ABB RAPID module: ReplayTargets_v11.mod

MODULE ReplayTargets_v11
    ! Generated from tests_v11.csv and success_v11.csv.
    ! Target names include testId. B* variants and configuration variables include testId and confId.

    ! Robtargets and jointtargets for replay
    CONST robtarget rA_t1 := [[1867.5,0,1823],[2.18557E-8,0,-1,0],[0,0,0,0],[9E+09,9E+09,9E+09,9E+09,9E+09,9E+09]];
    CONST robtarget rB_t1 := [[1165.98,1084.18,2334.34],[0.470302,-0.608433,0.138324,-0.624093],[0,3,3,0],[9E+09,9E+09,9E+09,9E+09,9E+09,9E+09]];
    CONST robtarget rB_t1_c5 := [[1165.98,1084.18,2334.34],[0.470302,-0.608433,0.138324,-0.624093],[0,0,0,0],[9E+09,9E+09,9E+09,9E+09,9E+09,9E+09]];
    CONST robtarget rB_t1_c6 := [[1165.98,1084.18,2334.34],[0.470302,-0.608433,0.138324,-0.624093],[0,4,0,0],[9E+09,9E+09,9E+09,9E+09,9E+09,9E+09]];
    CONST jointtarget jA_t1 := [[0,-2.3802E-6,7.25062E-7,0,90,0],[9E+09,9E+09,9E+09,9E+09,9E+09,9E+09]];
    CONST jointtarget jB_t1 := [[45.0004,-17.5512,3.9027,270,20.2686,315],[9E+09,9E+09,9E+09,9E+09,9E+09,9E+09]];
    CONST jointtarget jBseed_t1 := [[45.0004,-17.5512,3.9027,270,20.2686,315],[9E+09,9E+09,9E+09,9E+09,9E+09,9E+09]];

    CONST robtarget rA_t4 := [[-1793.05,1763.6,2052.64],[0.337402,0.281183,-0.557431,-0.704533],[1,-3,-1,0],[9E+09,9E+09,9E+09,9E+09,9E+09,9E+09]];
    CONST robtarget rB_t4 := [[-0.00867415,1613.24,1410.95],[0.623931,-0.332722,0.332726,0.623939],[1,-2,-2,0],[9E+09,9E+09,9E+09,9E+09,9E+09,9E+09]];
    CONST robtarget rB_t4_c1 := [[-0.00867415,1613.24,1410.95],[0.623931,-0.332722,0.332726,0.623939],[0,-4,-4,0],[9E+09,9E+09,9E+09,9E+09,9E+09,9E+09]];
    CONST robtarget rB_t4_c4 := [[-0.00867415,1613.24,1410.95],[0.623931,-0.332722,0.332726,0.623939],[0,-4,0,0],[9E+09,9E+09,9E+09,9E+09,9E+09,9E+09]];
    CONST jointtarget jA_t4 := [[134.999,27.2488,-32.8513,-225.001,10.1755,-45.0007],[9E+09,9E+09,9E+09,9E+09,9E+09,9E+09]];
    CONST jointtarget jB_t4 := [[90.0003,-18.1701,41.0059,-180,56.6967,-180],[9E+09,9E+09,9E+09,9E+09,9E+09,9E+09]];
    CONST jointtarget jBseed_t4 := [[90.0003,-18.1701,41.0059,-180,56.6967,-180],[9E+09,9E+09,9E+09,9E+09,9E+09,9E+09]];

    CONST robtarget rA_t7 := [[2738.04,83.3778,1374.99],[0.204279,-0.875639,-0.176726,-0.400366],[0,0,-3,0],[9E+09,9E+09,9E+09,9E+09,9E+09,9E+09]];
    CONST robtarget rB_t7 := [[2056.76,0.0250541,368.189],[0.572435,-0.30037,0.725174,-0.237103],[0,-2,-3,0],[9E+09,9E+09,9E+09,9E+09,9E+09,9E+09]];
    CONST robtarget rB_t7_c1 := [[2056.76,0.0250541,368.189],[0.572435,-0.30037,0.725174,-0.237103],[0,-4,-4,0],[9E+09,9E+09,9E+09,9E+09,9E+09,9E+09]];
    CONST robtarget rB_t7_c2 := [[2056.76,0.0250541,368.189],[0.572435,-0.30037,0.725174,-0.237103],[0,0,-4,0],[9E+09,9E+09,9E+09,9E+09,9E+09,9E+09]];
    CONST jointtarget jA_t7 := [[2.67622E-5,42.2346,-33.9622,45,44.9153,-225],[9E+09,9E+09,9E+09,9E+09,9E+09,9E+09]];
    CONST jointtarget jB_t7 := [[0.000739783,31.9694,26.4257,-179.999,44.9684,-224.999],[9E+09,9E+09,9E+09,9E+09,9E+09,9E+09]];
    CONST jointtarget jBseed_t7 := [[0.000739982,31.9694,26.4257,-179.999,44.9684,-224.999],[9E+09,9E+09,9E+09,9E+09,9E+09,9E+09]];

    CONST robtarget rA_t9 := [[-1368.98,-1368.96,2775.29],[0.617027,1.37404E-6,-0.488433,0.617018],[-2,-3,-4,0],[9E+09,9E+09,9E+09,9E+09,9E+09,9E+09]];
    CONST robtarget rB_t9 := [[-127.824,-1431.05,1500.85],[0.635695,0.309679,-0.685821,0.172164],[-2,-2,2,0],[9E+09,9E+09,9E+09,9E+09,9E+09,9E+09]];
    CONST robtarget rB_t9_c5 := [[-127.824,-1431.05,1500.85],[0.635695,0.309679,-0.685821,0.172164],[0,0,0,0],[9E+09,9E+09,9E+09,9E+09,9E+09,9E+09]];
    CONST jointtarget jA_t9 := [[-135,10.9152,-39.5999,-180,2.84006,-315],[9E+09,9E+09,9E+09,9E+09,9E+09,9E+09]];
    CONST jointtarget jB_t9 := [[-90.0007,-29.3912,41.2717,-90.0007,49.9344,269.999],[9E+09,9E+09,9E+09,9E+09,9E+09,9E+09]];
    CONST jointtarget jBseed_t9 := [[-90.0007,-29.3912,41.2717,-90.0007,49.9344,269.999],[9E+09,9E+09,9E+09,9E+09,9E+09,9E+09]];

    CONST robtarget rA_t12 := [[1027.41,1027.39,1309.98],[0.608549,-0.561103,0.561098,-7.84079E-6],[0,-3,1,0],[9E+09,9E+09,9E+09,9E+09,9E+09,9E+09]];
    CONST robtarget rB_t12 := [[-1587.99,1648.05,1389.04],[0.657658,-0.705427,-0.212225,0.15754],[1,-2,-4,0],[9E+09,9E+09,9E+09,9E+09,9E+09,9E+09]];
    CONST robtarget rB_t12_c4 := [[-1587.99,1648.05,1389.04],[0.657658,-0.705427,-0.212225,0.15754],[0,-4,0,0],[9E+09,9E+09,9E+09,9E+09,9E+09,9E+09]];
    CONST robtarget rB_t12_c5 := [[-1587.99,1648.05,1389.04],[0.657658,-0.705427,-0.212225,0.15754],[0,0,0,0],[9E+09,9E+09,9E+09,9E+09,9E+09,9E+09]];
    CONST jointtarget jA_t12 := [[44.9995,-30.1419,48.0401,-180.001,2.86752,134.999],[9E+09,9E+09,9E+09,9E+09,9E+09,9E+09]];
    CONST jointtarget jB_t12 := [[135,14.8265,5.47776,-135,21.0743,-315],[9E+09,9E+09,9E+09,9E+09,9E+09,9E+09]];
    CONST jointtarget jBseed_t12 := [[135,14.8265,5.47777,-135,21.0743,-315],[9E+09,9E+09,9E+09,9E+09,9E+09,9E+09]];

    CONST robtarget rA_t16 := [[-9.45088,2636.5,793.339],[0.463779,-0.798683,-0.345911,-0.165411],[0,-4,-3,0],[9E+09,9E+09,9E+09,9E+09,9E+09,9E+09]];
    CONST robtarget rB_t16 := [[1243.34,1193.68,2340.57],[0.833225,-0.325403,0.441958,-0.0672477],[0,-2,-3,0],[9E+09,9E+09,9E+09,9E+09,9E+09,9E+09]];
    CONST robtarget rB_t16_c2 := [[1243.34,1193.68,2340.57],[0.833225,-0.325403,0.441958,-0.0672477],[0,0,-4,0],[9E+09,9E+09,9E+09,9E+09,9E+09,9E+09]];
    CONST jointtarget jA_t16 := [[89.9999,41.6852,-10.6259,-270,3.24656,-225],[9E+09,9E+09,9E+09,9E+09,9E+09,9E+09]];
    CONST jointtarget jB_t16 := [[45.0001,-11.4243,-0.148013,-135,17.304,-270],[9E+09,9E+09,9E+09,9E+09,9E+09,9E+09]];
    CONST jointtarget jBseed_t16 := [[45.0001,-11.4243,-0.148018,-135,17.304,-270],[9E+09,9E+09,9E+09,9E+09,9E+09,9E+09]];

    CONST robtarget rA_t19 := [[-102.211,-1856.03,1361.59],[0.589306,0.574164,0.0334011,-0.567397],[-1,2,-2,0],[9E+09,9E+09,9E+09,9E+09,9E+09,9E+09]];
    CONST robtarget rB_t19 := [[1138.52,-1275.9,-60.9308],[0.259666,0.355191,0.770598,-0.461076],[-1,2,-3,0],[9E+09,9E+09,9E+09,9E+09,9E+09,9E+09]];
    CONST robtarget rB_t19_c2 := [[1138.52,-1275.9,-60.9308],[0.259666,0.355191,0.770598,-0.461076],[0,0,-4,0],[9E+09,9E+09,9E+09,9E+09,9E+09,9E+09]];
    CONST jointtarget jA_t19 := [[-89.9992,-3.43333,28.826,225.001,59.9707,-179.999],[9E+09,9E+09,9E+09,9E+09,9E+09,9E+09]];
    CONST jointtarget jB_t19 := [[-45.0008,43.0879,35.2809,224.999,55.327,-225.001],[9E+09,9E+09,9E+09,9E+09,9E+09,9E+09]];
    CONST jointtarget jBseed_t19 := [[-45.0008,43.0879,35.2809,224.999,55.327,-225.001],[9E+09,9E+09,9E+09,9E+09,9E+09,9E+09]];

    CONST robtarget rA_t22 := [[972.378,-908.4,1704.11],[0.389489,-0.323377,0.531814,-0.678896],[-1,1,-3,0],[9E+09,9E+09,9E+09,9E+09,9E+09,9E+09]];
    CONST robtarget rB_t22 := [[958.385,1131.9,1340.89],[0.368991,-0.50086,0.597944,0.505419],[0,0,2,0],[9E+09,9E+09,9E+09,9E+09,9E+09,9E+09]];
    CONST robtarget rB_t22_c5 := [[958.385,1131.9,1340.89],[0.368991,-0.50086,0.597944,0.505419],[0,0,0,0],[9E+09,9E+09,9E+09,9E+09,9E+09,9E+09]];
    CONST jointtarget jA_t22 := [[-45.0004,-38.8031,41.6208,135,22.53,-225],[9E+09,9E+09,9E+09,9E+09,9E+09,9E+09]];
    CONST jointtarget jB_t22 := [[44.9997,-25.3517,43.9894,89.9997,47.2848,270],[9E+09,9E+09,9E+09,9E+09,9E+09,9E+09]];
    CONST jointtarget jBseed_t22 := [[44.9997,-25.3517,43.9894,89.9997,47.2848,270],[9E+09,9E+09,9E+09,9E+09,9E+09,9E+09]];

    CONST robtarget rA_t23 := [[958.385,1131.9,1340.89],[0.368991,-0.50086,0.597944,0.505419],[0,0,2,0],[9E+09,9E+09,9E+09,9E+09,9E+09,9E+09]];
    CONST robtarget rB_t23 := [[-1885.02,1961.47,581.585],[0.429751,-0.871071,0.0769368,0.22501],[1,-2,-4,0],[9E+09,9E+09,9E+09,9E+09,9E+09,9E+09]];
    CONST robtarget rB_t23_c6 := [[-1885.02,1961.47,581.585],[0.429751,-0.871071,0.0769368,0.22501],[0,4,0,0],[9E+09,9E+09,9E+09,9E+09,9E+09,9E+09]];
    CONST jointtarget jA_t23 := [[44.9997,-25.3517,43.9894,89.9997,47.2848,270],[9E+09,9E+09,9E+09,9E+09,9E+09,9E+09]];
    CONST jointtarget jB_t23 := [[134.999,51.3205,-17.3031,-90.0009,18.8714,-315.001],[9E+09,9E+09,9E+09,9E+09,9E+09,9E+09]];
    CONST jointtarget jBseed_t23 := [[134.999,51.3205,-17.3031,-90.0009,18.8714,-315.001],[9E+09,9E+09,9E+09,9E+09,9E+09,9E+09]];

    CONST robtarget rA_t27 := [[-855.452,855.457,3218.91],[0.702987,0.107827,-1.23278E-6,0.702981],[1,1,1,0],[9E+09,9E+09,9E+09,9E+09,9E+09,9E+09]];
    CONST robtarget rB_t27 := [[0.00862806,893.795,2601.28],[0.375694,-0.0727351,-0.175609,-0.907042],[0,1,-1,0],[9E+09,9E+09,9E+09,9E+09,9E+09,9E+09]];
    CONST robtarget rB_t27_c5 := [[0.00862806,893.795,2601.28],[0.375694,-0.0727351,-0.175609,-0.907042],[0,0,0,0],[9E+09,9E+09,9E+09,9E+09,9E+09,9E+09]];
    CONST robtarget rB_t27_c8 := [[0.00862806,893.795,2601.28],[0.375694,-0.0727351,-0.175609,-0.907042],[0,0,4,0],[9E+09,9E+09,9E+09,9E+09,9E+09,9E+09]];
    CONST jointtarget jA_t27 := [[135,0.679351,-47.5347,180,55.5248,135],[9E+09,9E+09,9E+09,9E+09,9E+09,9E+09]];
    CONST jointtarget jB_t27 := [[89.9994,-41.2421,11.8296,179.999,38.673,-45.0006],[9E+09,9E+09,9E+09,9E+09,9E+09,9E+09]];
    CONST jointtarget jBseed_t27 := [[89.9994,-41.2421,11.8296,179.999,38.6731,-45.0006],[9E+09,9E+09,9E+09,9E+09,9E+09,9E+09]];

    CONST robtarget rA_t28 := [[0.00862806,893.795,2601.28],[0.375694,-0.0727351,-0.175609,-0.907042],[0,1,-1,0],[9E+09,9E+09,9E+09,9E+09,9E+09,9E+09]];
    CONST robtarget rB_t28 := [[66.616,1510.09,107.25],[0.0864039,-0.670046,-0.632294,-0.379179],[0,-2,3,0],[9E+09,9E+09,9E+09,9E+09,9E+09,9E+09]];
    CONST robtarget rB_t28_c5 := [[66.616,1510.09,107.25],[0.0864039,-0.670046,-0.632294,-0.379179],[0,0,0,0],[9E+09,9E+09,9E+09,9E+09,9E+09,9E+09]];
    CONST jointtarget jA_t28 := [[89.9994,-41.2421,11.8296,179.999,38.673,-45.0006],[9E+09,9E+09,9E+09,9E+09,9E+09,9E+09]];
    CONST jointtarget jB_t28 := [[89.9998,26.78,48.5241,-135,34.3388,315],[9E+09,9E+09,9E+09,9E+09,9E+09,9E+09]];
    CONST jointtarget jBseed_t28 := [[89.9998,26.78,48.5241,-135,34.3388,315],[9E+09,9E+09,9E+09,9E+09,9E+09,9E+09]];

    CONST robtarget rA_t31 := [[0.0247556,-2099.99,69.6706],[0.317201,0.631961,-0.63197,0.317209],[-1,-2,0,0],[9E+09,9E+09,9E+09,9E+09,9E+09,9E+09]];
    CONST robtarget rB_t31 := [[1527.9,-1527.94,1319.85],[0.854699,0.367072,0.36708,-1.01895E-5],[-1,1,-2,0],[9E+09,9E+09,9E+09,9E+09,9E+09,9E+09]];
    CONST robtarget rB_t31_c1 := [[1527.9,-1527.94,1319.85],[0.854699,0.367072,0.36708,-1.01895E-5],[0,-4,-4,0],[9E+09,9E+09,9E+09,9E+09,9E+09,9E+09]];
    CONST robtarget rB_t31_c4 := [[1527.9,-1527.94,1319.85],[0.854699,0.367072,0.36708,-1.01895E-5],[0,-4,0,0],[9E+09,9E+09,9E+09,9E+09,9E+09,9E+09]];
    CONST jointtarget jA_t31 := [[-89.9993,44.4173,19.4034,-179.999,27.1279,0.000700849],[9E+09,9E+09,9E+09,9E+09,9E+09,9E+09]];
    CONST jointtarget jB_t31 := [[-45.0007,11.4902,15.5232,179.999,54.4664,-135.001],[9E+09,9E+09,9E+09,9E+09,9E+09,9E+09]];
    CONST jointtarget jBseed_t31 := [[-45.0007,11.4902,15.5232,179.999,54.4664,-135.001],[9E+09,9E+09,9E+09,9E+09,9E+09,9E+09]];

    CONST robtarget rA_t37 := [[-1966.29,1997.86,669.131],[0.118201,0.309457,-0.836468,-0.436563],[1,-1,1,0],[9E+09,9E+09,9E+09,9E+09,9E+09,9E+09]];
    CONST robtarget rB_t37 := [[2614.3,138.194,1907.14],[0.237671,0.177553,0.665957,0.684463],[0,1,4,0],[9E+09,9E+09,9E+09,9E+09,9E+09,9E+09]];
    CONST robtarget rB_t37_c5 := [[2614.3,138.194,1907.14],[0.237671,0.177553,0.665957,0.684463],[0,0,0,0],[9E+09,9E+09,9E+09,9E+09,9E+09,9E+09]];
    CONST jointtarget jA_t37 := [[135.001,53.3164,-24.4761,-44.9994,10.9098,135.001],[9E+09,9E+09,9E+09,9E+09,9E+09,9E+09]];
    CONST jointtarget jB_t37 := [[0.000991918,37.2063,-42.3057,90.001,55.8159,360.001],[9E+09,9E+09,9E+09,9E+09,9E+09,9E+09]];
    CONST jointtarget jBseed_t37 := [[0.000991821,37.2063,-42.3057,90.001,55.8159,360.001],[9E+09,9E+09,9E+09,9E+09,9E+09,9E+09]];

    CONST robtarget rA_t40 := [[2042.82,2042.82,1269.08],[2.13329E-8,0.491803,0.491803,0.718512],[0,2,3,0],[9E+09,9E+09,9E+09,9E+09,9E+09,9E+09]];
    CONST robtarget rB_t40 := [[2226.68,51.0258,2546.48],[0.890874,-0.128724,0.42641,0.0891495],[0,-3,-2,0],[9E+09,9E+09,9E+09,9E+09,9E+09,9E+09]];
    CONST robtarget rB_t40_c8 := [[2226.68,51.0258,2546.48],[0.890874,-0.128724,0.42641,0.0891495],[0,0,4,0],[9E+09,9E+09,9E+09,9E+09,9E+09,9E+09]];
    CONST jointtarget jA_t40 := [[45,49.2001,-36.7553,180,14.3083,315],[9E+09,9E+09,9E+09,9E+09,9E+09,9E+09]];
    CONST jointtarget jB_t40 := [[0.000737447,21.2244,-41.8256,-224.999,25.5861,-134.999],[9E+09,9E+09,9E+09,9E+09,9E+09,9E+09]];
    CONST jointtarget jBseed_t40 := [[0.00073748,21.2244,-41.8256,-224.999,25.5861,-134.999],[9E+09,9E+09,9E+09,9E+09,9E+09,9E+09]];

    CONST robtarget rA_t46 := [[315.105,315.107,2762.98],[0.664534,5.18351E-7,0.341732,0.66454],[0,-2,-2,0],[9E+09,9E+09,9E+09,9E+09,9E+09,9E+09]];
    CONST robtarget rB_t46 := [[1363.27,1399.66,1627.46],[0.295621,-0.697087,-0.341342,-0.556923],[0,-3,-3,0],[9E+09,9E+09,9E+09,9E+09,9E+09,9E+09]];
    CONST robtarget rB_t46_c1 := [[1363.27,1399.66,1627.46],[0.295621,-0.697087,-0.341342,-0.556923],[0,-4,-4,0],[9E+09,9E+09,9E+09,9E+09,9E+09,9E+09]];
    CONST robtarget rB_t46_c2 := [[1363.27,1399.66,1627.46],[0.295621,-0.697087,-0.341342,-0.556923],[0,0,-4,0],[9E+09,9E+09,9E+09,9E+09,9E+09,9E+09]];
    CONST jointtarget jA_t46 := [[45.0002,-51.9395,4.53749,-180,2.63314,-135],[9E+09,9E+09,9E+09,9E+09,9E+09,9E+09]];
    CONST jointtarget jB_t46 := [[45.0007,-4.25367,16.2215,-269.999,8.85525,-269.999],[9E+09,9E+09,9E+09,9E+09,9E+09,9E+09]];
    CONST jointtarget jBseed_t46 := [[45.0007,-4.25367,16.2215,-269.999,8.85525,-269.999],[9E+09,9E+09,9E+09,9E+09,9E+09,9E+09]];

    CONST robtarget rA_t50 := [[-1650.69,1788.89,2235.47],[0.742108,-0.354072,-0.189288,-0.53673],[1,-2,3,0],[9E+09,9E+09,9E+09,9E+09,9E+09,9E+09]];
    CONST robtarget rB_t50 := [[44.2638,306.55,3391.36],[0.355804,-0.140867,0.00668765,-0.923859],[0,2,-2,0],[9E+09,9E+09,9E+09,9E+09,9E+09,9E+09]];
    CONST robtarget rB_t50_c7 := [[44.2638,306.55,3391.36],[0.355804,-0.140867,0.00668765,-0.923859],[0,-4,4,0],[9E+09,9E+09,9E+09,9E+09,9E+09,9E+09]];
    CONST jointtarget jA_t50 := [[135.001,29.556,-40.0324,-134.999,55.8782,315.001],[9E+09,9E+09,9E+09,9E+09,9E+09,9E+09]];
    CONST jointtarget jB_t50 := [[89.9996,-20.9717,-47.8442,225,22.0136,-90.0004],[9E+09,9E+09,9E+09,9E+09,9E+09,9E+09]];
    CONST jointtarget jBseed_t50 := [[89.9996,-20.9717,-47.8442,225,22.0136,-90.0004],[9E+09,9E+09,9E+09,9E+09,9E+09,9E+09]];

    CONST robtarget rA_t51 := [[44.2638,306.55,3391.36],[0.355804,-0.140867,0.00668765,-0.923859],[0,2,-2,0],[9E+09,9E+09,9E+09,9E+09,9E+09,9E+09]];
    CONST robtarget rB_t51 := [[2033.92,45.4637,1419.42],[0.577235,0.205402,0.70222,0.362625],[0,1,-1,0],[9E+09,9E+09,9E+09,9E+09,9E+09,9E+09]];
    CONST robtarget rB_t51_c5 := [[2033.92,45.4637,1419.42],[0.577235,0.205402,0.70222,0.362625],[0,0,0,0],[9E+09,9E+09,9E+09,9E+09,9E+09,9E+09]];
    CONST robtarget rB_t51_c8 := [[2033.92,45.4637,1419.42],[0.577235,0.205402,0.70222,0.362625],[0,0,4,0],[9E+09,9E+09,9E+09,9E+09,9E+09,9E+09]];
    CONST jointtarget jA_t51 := [[89.9996,-20.9717,-47.8442,225,22.0136,-90.0004],[9E+09,9E+09,9E+09,9E+09,9E+09,9E+09]];
    CONST jointtarget jB_t51 := [[0.000420681,1.789,18.8479,135,22.6362,-89.9996],[9E+09,9E+09,9E+09,9E+09,9E+09,9E+09]];
    CONST jointtarget jBseed_t51 := [[0.000420515,1.789,18.8479,135,22.6362,-89.9996],[9E+09,9E+09,9E+09,9E+09,9E+09,9E+09]];

    CONST robtarget rA_t53 := [[39.7549,2396.44,2309.29],[0.688612,-0.598908,0.352715,0.206675],[1,-1,-4,0],[9E+09,9E+09,9E+09,9E+09,9E+09,9E+09]];
    CONST robtarget rB_t53 := [[1503.67,-0.0118296,1707.84],[0.639783,0.276074,0.666511,0.264998],[-1,1,-2,0],[9E+09,9E+09,9E+09,9E+09,9E+09,9E+09]];
    CONST robtarget rB_t53_c1 := [[1503.67,-0.0118296,1707.84],[0.639783,0.276074,0.666511,0.264998],[0,-4,-4,0],[9E+09,9E+09,9E+09,9E+09,9E+09,9E+09]];
    CONST jointtarget jA_t53 := [[90.0007,25.6044,-41.7978,-44.9993,19.6881,-359.999],[9E+09,9E+09,9E+09,9E+09,9E+09,9E+09]];
    CONST jointtarget jB_t53 := [[-0.000453216,-28.9554,33.9439,180,2.64412,-135],[9E+09,9E+09,9E+09,9E+09,9E+09,9E+09]];
    CONST jointtarget jBseed_t53 := [[-0.000453108,-28.9554,33.9439,180,2.64412,-135],[9E+09,9E+09,9E+09,9E+09,9E+09,9E+09]];

    CONST robtarget rA_t56 := [[-781.455,-757.26,2911.76],[0.356269,-0.225306,-0.422891,0.802167],[-2,-1,-1,0],[9E+09,9E+09,9E+09,9E+09,9E+09,9E+09]];
    CONST robtarget rB_t56 := [[-1461,-1377.29,2942.46],[0.626638,0.215306,-0.16846,-0.729787],[-2,2,2,0],[9E+09,9E+09,9E+09,9E+09,9E+09,9E+09]];
    CONST robtarget rB_t56_c2 := [[-1461,-1377.29,2942.46],[0.626638,0.215306,-0.16846,-0.729787],[0,0,-4,0],[9E+09,9E+09,9E+09,9E+09,9E+09,9E+09]];
    CONST robtarget rB_t56_c5 := [[-1461,-1377.29,2942.46],[0.626638,0.215306,-0.16846,-0.729787],[0,0,0,0],[9E+09,9E+09,9E+09,9E+09,9E+09,9E+09]];
    CONST jointtarget jA_t56 := [[-135,-23.7587,-15.0853,-45.0001,8.32972,-45.0001],[9E+09,9E+09,9E+09,9E+09,9E+09,9E+09]];
    CONST jointtarget jB_t56 := [[-134.999,34.2473,-77.4173,225.001,30.0943,180.001],[9E+09,9E+09,9E+09,9E+09,9E+09,9E+09]];
    CONST jointtarget jBseed_t56 := [[-134.999,34.2473,-77.4172,225.001,30.0943,180.001],[9E+09,9E+09,9E+09,9E+09,9E+09,9E+09]];

    CONST robtarget rA_t58 := [[-516.819,-387.904,3130.9],[0.270635,0.128291,-0.254314,-0.919578],[-2,2,1,0],[9E+09,9E+09,9E+09,9E+09,9E+09,9E+09]];
    CONST robtarget rB_t58 := [[18.5522,-2972.36,1606.68],[0.550399,0.443924,0.502249,-0.497733],[-1,1,-1,0],[9E+09,9E+09,9E+09,9E+09,9E+09,9E+09]];
    CONST robtarget rB_t58_c8 := [[18.5522,-2972.36,1606.68],[0.550399,0.443924,0.502249,-0.497733],[0,0,4,0],[9E+09,9E+09,9E+09,9E+09,9E+09,9E+09]];
    CONST jointtarget jA_t58 := [[-135.001,-26.8752,-23.6708,224.999,50.524,134.999],[9E+09,9E+09,9E+09,9E+09,9E+09,9E+09]];
    CONST jointtarget jB_t58 := [[-89.9996,59.8242,-65.6776,90.0005,6.37043,-89.9997],[9E+09,9E+09,9E+09,9E+09,9E+09,9E+09]];
    CONST jointtarget jBseed_t58 := [[-89.9996,59.8242,-65.6777,90.0004,6.37043,-89.9996],[9E+09,9E+09,9E+09,9E+09,9E+09,9E+09]];

    CONST robtarget rA_t64 := [[-1515.54,1515.56,1455.6],[0.333635,0.187434,-0.452494,-0.805485],[1,-3,-2,0],[9E+09,9E+09,9E+09,9E+09,9E+09,9E+09]];
    CONST robtarget rB_t64 := [[2573.98,0.0267315,1917.9],[1.18647E-5,-0.542748,4.45635E-6,-0.839896],[0,-2,4,0],[9E+09,9E+09,9E+09,9E+09,9E+09,9E+09]];
    CONST robtarget rB_t64_c4 := [[2573.98,0.0267315,1917.9],[1.18647E-5,-0.542748,4.45635E-6,-0.839896],[0,-4,0,0],[9E+09,9E+09,9E+09,9E+09,9E+09,9E+09]];
    CONST jointtarget jA_t64 := [[135,8.96329,13.5435,-180,53.8548,-90.0005],[9E+09,9E+09,9E+09,9E+09,9E+09,9E+09]];
    CONST jointtarget jB_t64 := [[0.000611133,29.7098,-29.9512,-179.999,24.0168,360.001],[9E+09,9E+09,9E+09,9E+09,9E+09,9E+09]];
    CONST jointtarget jBseed_t64 := [[0.000611133,29.7098,-29.9512,-179.999,24.0168,360.001],[9E+09,9E+09,9E+09,9E+09,9E+09,9E+09]];

    CONST robtarget rA_t66 := [[2907.11,71.3398,1111.81],[0.299575,0.451234,0.640506,0.544421],[0,-3,4,0],[9E+09,9E+09,9E+09,9E+09,9E+09,9E+09]];
    CONST robtarget rB_t66 := [[1282.21,1138.81,-182.246],[0.536967,0.025283,0.842048,0.0445313],[0,-2,-3,0],[9E+09,9E+09,9E+09,9E+09,9E+09,9E+09]];
    CONST robtarget rB_t66_c4 := [[1282.21,1138.81,-182.246],[0.536967,0.025283,0.842048,0.0445313],[0,-4,0,0],[9E+09,9E+09,9E+09,9E+09,9E+09,9E+09]];
    CONST jointtarget jA_t66 := [[0.000451427,52.8733,-38.2867,-270,25.2803,360],[9E+09,9E+09,9E+09,9E+09,9E+09,9E+09]];
    CONST jointtarget jB_t66 := [[45,49.9838,31.7103,-135,59.1723,-180],[9E+09,9E+09,9E+09,9E+09,9E+09,9E+09]];
    CONST jointtarget jBseed_t66 := [[45,49.9838,31.7103,-135,59.1723,-180],[9E+09,9E+09,9E+09,9E+09,9E+09,9E+09]];

    CONST robtarget rA_t67 := [[1282.21,1138.81,-182.246],[0.536967,0.025283,0.842048,0.0445313],[0,-2,-3,0],[9E+09,9E+09,9E+09,9E+09,9E+09,9E+09]];
    CONST robtarget rB_t67 := [[33.2258,843.078,3012.65],[0.865057,-0.313323,0.22989,0.317263],[0,-2,-4,0],[9E+09,9E+09,9E+09,9E+09,9E+09,9E+09]];
    CONST robtarget rB_t67_c2 := [[33.2258,843.078,3012.65],[0.865057,-0.313323,0.22989,0.317263],[0,0,-4,0],[9E+09,9E+09,9E+09,9E+09,9E+09,9E+09]];
    CONST robtarget rB_t67_c3 := [[33.2258,843.078,3012.65],[0.865057,-0.313323,0.22989,0.317263],[0,4,-4,0],[9E+09,9E+09,9E+09,9E+09,9E+09,9E+09]];
    CONST jointtarget jA_t67 := [[45,49.9838,31.7103,-135,59.1723,-180],[9E+09,9E+09,9E+09,9E+09,9E+09,9E+09]];
    CONST jointtarget jB_t67 := [[89.9996,-28.5745,-16.8389,-90.0004,11.4737,-315],[9E+09,9E+09,9E+09,9E+09,9E+09,9E+09]];
    CONST jointtarget jBseed_t67 := [[89.9996,-28.5745,-16.8389,-90.0004,11.4737,-315],[9E+09,9E+09,9E+09,9E+09,9E+09,9E+09]];

    CONST robtarget rA_t68 := [[33.2258,843.078,3012.65],[0.865057,-0.313323,0.22989,0.317263],[0,-2,-4,0],[9E+09,9E+09,9E+09,9E+09,9E+09,9E+09]];
    CONST robtarget rB_t68 := [[1863.94,-1731.5,1359.6],[0.365907,0.552226,0.180387,0.727062],[-1,-3,-1,0],[9E+09,9E+09,9E+09,9E+09,9E+09,9E+09]];
    CONST robtarget rB_t68_c4 := [[1863.94,-1731.5,1359.6],[0.365907,0.552226,0.180387,0.727062],[0,-4,0,0],[9E+09,9E+09,9E+09,9E+09,9E+09,9E+09]];
    CONST jointtarget jA_t68 := [[89.9996,-28.5745,-16.8389,-90.0004,11.4737,-315],[9E+09,9E+09,9E+09,9E+09,9E+09,9E+09]];
    CONST jointtarget jB_t68 := [[-45.0004,30.585,-11.0544,-225,52.4851,-0.000424009],[9E+09,9E+09,9E+09,9E+09,9E+09,9E+09]];
    CONST jointtarget jBseed_t68 := [[-45.0004,30.585,-11.0544,-225,52.4851,-0.00042436],[9E+09,9E+09,9E+09,9E+09,9E+09,9E+09]];

    CONST robtarget rA_t69 := [[1863.94,-1731.5,1359.6],[0.365907,0.552226,0.180387,0.727062],[-1,-3,-1,0],[9E+09,9E+09,9E+09,9E+09,9E+09,9E+09]];
    CONST robtarget rB_t69 := [[90.2483,-604.038,3447.57],[0.635996,0.309007,0.0836555,0.702158],[-1,1,-3,0],[9E+09,9E+09,9E+09,9E+09,9E+09,9E+09]];
    CONST robtarget rB_t69_c4 := [[90.2483,-604.038,3447.57],[0.635996,0.309007,0.0836555,0.702158],[0,-4,0,0],[9E+09,9E+09,9E+09,9E+09,9E+09,9E+09]];
    CONST jointtarget jA_t69 := [[-45.0004,30.585,-11.0544,-225,52.4851,-0.000424009],[9E+09,9E+09,9E+09,9E+09,9E+09,9E+09]];
    CONST jointtarget jB_t69 := [[-89.999,-4.08885,-66.7925,90.001,32.7073,-269.999],[9E+09,9E+09,9E+09,9E+09,9E+09,9E+09]];
    CONST jointtarget jBseed_t69 := [[-89.999,-4.08887,-66.7925,90.001,32.7073,-269.999],[9E+09,9E+09,9E+09,9E+09,9E+09,9E+09]];

    CONST robtarget rA_t72 := [[72.5438,-307.938,3482.9],[0.882145,-0.0280946,0.25871,0.392555],[-1,-3,4,0],[9E+09,9E+09,9E+09,9E+09,9E+09,9E+09]];
    CONST robtarget rB_t72 := [[-1617.38,-1478.51,2678.01],[0.645209,0.274316,-0.69781,-0.14669],[-2,-1,2,0],[9E+09,9E+09,9E+09,9E+09,9E+09,9E+09]];
    CONST robtarget rB_t72_c5 := [[-1617.38,-1478.51,2678.01],[0.645209,0.274316,-0.69781,-0.14669],[0,0,0,0],[9E+09,9E+09,9E+09,9E+09,9E+09,9E+09]];
    CONST jointtarget jA_t72 := [[-89.9997,-5.67095,-71.7875,-225,37.9022,360],[9E+09,9E+09,9E+09,9E+09,9E+09,9E+09]];
    CONST jointtarget jB_t72 := [[-135,34.5695,-72.3707,-44.9996,56.2737,180],[9E+09,9E+09,9E+09,9E+09,9E+09,9E+09]];
    CONST jointtarget jBseed_t72 := [[-135,34.5695,-72.3707,-44.9996,56.2737,180],[9E+09,9E+09,9E+09,9E+09,9E+09,9E+09]];

    CONST robtarget rA_t73 := [[-1617.38,-1478.51,2678.01],[0.645209,0.274316,-0.69781,-0.14669],[-2,-1,2,0],[9E+09,9E+09,9E+09,9E+09,9E+09,9E+09]];
    CONST robtarget rB_t73 := [[1512.76,1682.59,2148.43],[0.670669,-0.609575,-0.292732,-0.304844],[0,0,-3,0],[9E+09,9E+09,9E+09,9E+09,9E+09,9E+09]];
    CONST robtarget rB_t73_c4 := [[1512.76,1682.59,2148.43],[0.670669,-0.609575,-0.292732,-0.304844],[0,-4,0,0],[9E+09,9E+09,9E+09,9E+09,9E+09,9E+09]];
    CONST jointtarget jA_t73 := [[-135,34.5695,-72.3707,-44.9996,56.2737,180],[9E+09,9E+09,9E+09,9E+09,9E+09,9E+09]];
    CONST jointtarget jB_t73 := [[44.9995,16.2365,-23.3018,89.9995,45.9902,-225.001],[9E+09,9E+09,9E+09,9E+09,9E+09,9E+09]];
    CONST jointtarget jBseed_t73 := [[44.9995,16.2365,-23.3018,89.9995,45.9902,-225.001],[9E+09,9E+09,9E+09,9E+09,9E+09,9E+09]];

    CONST robtarget rA_t74 := [[1512.76,1682.59,2148.43],[0.670669,-0.609575,-0.292732,-0.304844],[0,0,-3,0],[9E+09,9E+09,9E+09,9E+09,9E+09,9E+09]];
    CONST robtarget rB_t74 := [[1174.89,-1292.72,-255.154],[0.430425,0.901012,-0.0205942,0.0498761],[-1,-2,-2,0],[9E+09,9E+09,9E+09,9E+09,9E+09,9E+09]];
    CONST robtarget rB_t74_c4 := [[1174.89,-1292.72,-255.154],[0.430425,0.901012,-0.0205942,0.0498761],[0,-4,0,0],[9E+09,9E+09,9E+09,9E+09,9E+09,9E+09]];
    CONST jointtarget jA_t74 := [[44.9995,16.2365,-23.3018,89.9995,45.9902,-225.001],[9E+09,9E+09,9E+09,9E+09,9E+09,9E+09]];
    CONST jointtarget jB_t74 := [[-45.0001,52.7342,28.5125,-135,44.8732,-90.0001],[9E+09,9E+09,9E+09,9E+09,9E+09,9E+09]];
    CONST jointtarget jBseed_t74 := [[-45.0001,52.7342,28.5125,-135,44.8732,-90.0001],[9E+09,9E+09,9E+09,9E+09,9E+09,9E+09]];

    CONST robtarget rA_t79 := [[-816.378,919.561,-368.344],[0.272348,-0.894319,0.350624,0.0555271],[1,-2,-3,0],[9E+09,9E+09,9E+09,9E+09,9E+09,9E+09]];
    CONST robtarget rB_t79 := [[-881.287,1006.84,2597.32],[0.918162,-0.360497,-0.0185053,-0.163334],[1,-2,-5,0],[9E+09,9E+09,9E+09,9E+09,9E+09,9E+09]];
    CONST robtarget rB_t79_c1 := [[-881.287,1006.84,2597.32],[0.918162,-0.360497,-0.0185053,-0.163334],[0,-4,-4,0],[9E+09,9E+09,9E+09,9E+09,9E+09,9E+09]];
    CONST robtarget rB_t79_c4 := [[-881.287,1006.84,2597.32],[0.918162,-0.360497,-0.0185053,-0.163334],[0,-4,0,0],[9E+09,9E+09,9E+09,9E+09,9E+09,9E+09]];
    CONST jointtarget jA_t79 := [[134.999,53.7339,45.3502,-135.001,38.1512,-225.001],[9E+09,9E+09,9E+09,9E+09,9E+09,9E+09]];
    CONST jointtarget jB_t79 := [[135,-21.7334,-0.195621,-135,48.7478,-360],[9E+09,9E+09,9E+09,9E+09,9E+09,9E+09]];
    CONST jointtarget jBseed_t79 := [[135,-21.7334,-0.195625,-135,48.7478,-360],[9E+09,9E+09,9E+09,9E+09,9E+09,9E+09]];

    CONST robtarget rA_t82 := [[-206.925,281.712,3308.39],[0.337776,-0.0648298,-0.253186,-0.904213],[1,3,2,0],[9E+09,9E+09,9E+09,9E+09,9E+09,9E+09]];
    CONST robtarget rB_t82 := [[-869.622,1036.66,1582.29],[0.613039,-0.668325,-0.309037,-0.286392],[1,-1,-1,0],[9E+09,9E+09,9E+09,9E+09,9E+09,9E+09]];
    CONST robtarget rB_t82_c8 := [[-869.622,1036.66,1582.29],[0.613039,-0.668325,-0.309037,-0.286392],[0,0,4,0],[9E+09,9E+09,9E+09,9E+09,9E+09,9E+09]];
    CONST robtarget rB_t82_c9 := [[-869.622,1036.66,1582.29],[0.613039,-0.668325,-0.309037,-0.286392],[0,4,4,0],[9E+09,9E+09,9E+09,9E+09,9E+09,9E+09]];
    CONST jointtarget jA_t82 := [[135.001,-26.4467,-39.0921,270.001,18.4631,180.001],[9E+09,9E+09,9E+09,9E+09,9E+09,9E+09]];
    CONST jointtarget jB_t82 := [[135.001,-35.4485,42.2993,-89.9994,45.0197,-44.9994],[9E+09,9E+09,9E+09,9E+09,9E+09,9E+09]];
    CONST jointtarget jBseed_t82 := [[135.001,-35.4485,42.2993,-89.9994,45.0197,-44.9994],[9E+09,9E+09,9E+09,9E+09,9E+09,9E+09]];

    CONST robtarget rA_t83 := [[-869.622,1036.66,1582.29],[0.613039,-0.668325,-0.309037,-0.286392],[1,-1,-1,0],[9E+09,9E+09,9E+09,9E+09,9E+09,9E+09]];
    CONST robtarget rB_t83 := [[-1630.62,1808.91,1755.18],[0.218749,-0.280556,-0.670403,-0.651151],[1,-1,-2,0],[9E+09,9E+09,9E+09,9E+09,9E+09,9E+09]];
    CONST robtarget rB_t83_c5 := [[-1630.62,1808.91,1755.18],[0.218749,-0.280556,-0.670403,-0.651151],[0,0,0,0],[9E+09,9E+09,9E+09,9E+09,9E+09,9E+09]];
    CONST robtarget rB_t83_c8 := [[-1630.62,1808.91,1755.18],[0.218749,-0.280556,-0.670403,-0.651151],[0,0,4,0],[9E+09,9E+09,9E+09,9E+09,9E+09,9E+09]];
    CONST jointtarget jA_t83 := [[135.001,-35.4485,42.2993,-89.9994,45.0197,-44.9994],[9E+09,9E+09,9E+09,9E+09,9E+09,9E+09]];
    CONST jointtarget jB_t83 := [[135.001,23.3595,-18.4338,-89.9991,49.0353,-134.999],[9E+09,9E+09,9E+09,9E+09,9E+09,9E+09]];
    CONST jointtarget jBseed_t83 := [[135.001,23.3595,-18.4338,-89.9991,49.0353,-134.999],[9E+09,9E+09,9E+09,9E+09,9E+09,9E+09]];

    CONST robtarget rA_t85 := [[1930.15,55.1772,809.731],[0.437101,-0.407513,0.801635,-0.0160386],[-1,-4,2,0],[9E+09,9E+09,9E+09,9E+09,9E+09,9E+09]];
    CONST robtarget rB_t85 := [[1483.71,-1619.15,2708.51],[0.145458,0.140219,-0.512339,0.834679],[-1,-1,3,0],[9E+09,9E+09,9E+09,9E+09,9E+09,9E+09]];
    CONST robtarget rB_t85_c8 := [[1483.71,-1619.15,2708.51],[0.145458,0.140219,-0.512339,0.834679],[0,0,4,0],[9E+09,9E+09,9E+09,9E+09,9E+09,9E+09]];
    CONST jointtarget jA_t85 := [[-0.000696811,9.747,31.1072,-270.001,19.3017,224.999],[9E+09,9E+09,9E+09,9E+09,9E+09,9E+09]];
    CONST jointtarget jB_t85 := [[-44.9998,29.6512,-61.7817,-89.9998,34.9944,315],[9E+09,9E+09,9E+09,9E+09,9E+09,9E+09]];
    CONST jointtarget jBseed_t85 := [[-44.9998,29.6512,-61.7817,-89.9998,34.9944,315],[9E+09,9E+09,9E+09,9E+09,9E+09,9E+09]];

    CONST robtarget rA_t88 := [[1883.97,-1693.67,1011.01],[0.601852,-0.23589,0.760816,-0.0573519],[-1,-4,2,0],[9E+09,9E+09,9E+09,9E+09,9E+09,9E+09]];
    CONST robtarget rB_t88 := [[2631.34,-134.594,1793.98],[0.673616,0.670251,0.215022,0.225323],[0,3,-2,0],[9E+09,9E+09,9E+09,9E+09,9E+09,9E+09]];
    CONST robtarget rB_t88_c5 := [[2631.34,-134.594,1793.98],[0.673616,0.670251,0.215022,0.225323],[0,0,0,0],[9E+09,9E+09,9E+09,9E+09,9E+09,9E+09]];
    CONST jointtarget jA_t88 := [[-45,35.6096,-8.59859,-270,53.6845,225],[9E+09,9E+09,9E+09,9E+09,9E+09,9E+09]];
    CONST jointtarget jB_t88 := [[0.000497925,36.6314,-37.5091,270,53.7156,-179.999],[9E+09,9E+09,9E+09,9E+09,9E+09,9E+09]];
    CONST jointtarget jBseed_t88 := [[0.000497909,36.6314,-37.5091,270,53.7156,-179.999],[9E+09,9E+09,9E+09,9E+09,9E+09,9E+09]];

    CONST robtarget rA_t89 := [[2631.34,-134.594,1793.98],[0.673616,0.670251,0.215022,0.225323],[0,3,-2,0],[9E+09,9E+09,9E+09,9E+09,9E+09,9E+09]];
    CONST robtarget rB_t89 := [[-0.0100308,-1992.85,2351.79],[0.79034,0.612668,1.64E-6,-5.9405E-6],[-2,-3,-2,0],[9E+09,9E+09,9E+09,9E+09,9E+09,9E+09]];
    CONST robtarget rB_t89_c5 := [[-0.0100308,-1992.85,2351.79],[0.79034,0.612668,1.64E-6,-5.9405E-6],[0,0,0,0],[9E+09,9E+09,9E+09,9E+09,9E+09,9E+09]];
    CONST jointtarget jA_t89 := [[0.000497925,36.6314,-37.5091,270,53.7156,-179.999],[9E+09,9E+09,9E+09,9E+09,9E+09,9E+09]];
    CONST jointtarget jB_t89 := [[-90.0003,2.06001,-14.1966,-180,2.29804,-90.0003],[9E+09,9E+09,9E+09,9E+09,9E+09,9E+09]];
    CONST jointtarget jBseed_t89 := [[-90.0003,2.06,-14.1966,-180,2.29804,-90.0003],[9E+09,9E+09,9E+09,9E+09,9E+09,9E+09]];

    CONST robtarget rA_t90 := [[-0.0100308,-1992.85,2351.79],[0.79034,0.612668,1.64E-6,-5.9405E-6],[-2,-3,-2,0],[9E+09,9E+09,9E+09,9E+09,9E+09,9E+09]];
    CONST robtarget rB_t90 := [[1939.65,1939.58,1900.24],[0.407797,-0.829006,0.343384,-0.168931],[0,-1,2,0],[9E+09,9E+09,9E+09,9E+09,9E+09,9E+09]];
    CONST robtarget rB_t90_c5 := [[1939.65,1939.58,1900.24],[0.407797,-0.829006,0.343384,-0.168931],[0,0,0,0],[9E+09,9E+09,9E+09,9E+09,9E+09,9E+09]];
    CONST jointtarget jA_t90 := [[-90.0003,2.06001,-14.1966,-180,2.29804,-90.0003],[9E+09,9E+09,9E+09,9E+09,9E+09,9E+09]];
    CONST jointtarget jB_t90 := [[44.9991,49.6066,-65.1103,-0.000908008,53.1168,269.999],[9E+09,9E+09,9E+09,9E+09,9E+09,9E+09]];
    CONST jointtarget jBseed_t90 := [[44.9991,49.6066,-65.1103,-0.000909421,53.1169,269.999],[9E+09,9E+09,9E+09,9E+09,9E+09,9E+09]];

    CONST robtarget rA_t102 := [[-1948.31,-1917.18,1251.26],[0.646342,0.509608,-0.56543,-0.053206],[-2,2,-1,0],[9E+09,9E+09,9E+09,9E+09,9E+09,9E+09]];
    CONST robtarget rB_t102 := [[-8.1709,-1803.03,1617.76],[0.576867,0.721357,0.282027,-0.259478],[-1,-1,1,0],[9E+09,9E+09,9E+09,9E+09,9E+09,9E+09]];
    CONST robtarget rB_t102_c3 := [[-8.1709,-1803.03,1617.76],[0.576867,0.721357,0.282027,-0.259478],[0,4,-4,0],[9E+09,9E+09,9E+09,9E+09,9E+09,9E+09]];
    CONST jointtarget jA_t102 := [[-135,39.4037,-22.5361,225,10.7523,-89.9997],[9E+09,9E+09,9E+09,9E+09,9E+09,9E+09]];
    CONST jointtarget jB_t102 := [[-89.9998,-12.197,23.7358,-89.9998,2.80709,135],[9E+09,9E+09,9E+09,9E+09,9E+09,9E+09]];
    CONST jointtarget jBseed_t102 := [[-89.9998,-12.197,23.7358,-89.9998,2.80709,135],[9E+09,9E+09,9E+09,9E+09,9E+09,9E+09]];

    CONST robtarget rA_t103 := [[-8.1709,-1803.03,1617.76],[0.576867,0.721357,0.282027,-0.259478],[-1,-1,1,0],[9E+09,9E+09,9E+09,9E+09,9E+09,9E+09]];
    CONST robtarget rB_t103 := [[2153.31,0.0367459,1279.08],[0.0943866,0.700781,0.700775,0.0943998],[0,0,-3,0],[9E+09,9E+09,9E+09,9E+09,9E+09,9E+09]];
    CONST robtarget rB_t103_c5 := [[2153.31,0.0367459,1279.08],[0.0943866,0.700781,0.700775,0.0943998],[0,0,0,0],[9E+09,9E+09,9E+09,9E+09,9E+09,9E+09]];
    CONST jointtarget jA_t103 := [[-89.9998,-12.197,23.7358,-89.9998,2.80709,135],[9E+09,9E+09,9E+09,9E+09,9E+09,9E+09]];
    CONST jointtarget jB_t103 := [[0.00091901,13.5118,5.64439,0.000918909,55.501,-269.999],[9E+09,9E+09,9E+09,9E+09,9E+09,9E+09]];
    CONST jointtarget jBseed_t103 := [[0.000919004,13.5118,5.64439,0.000919004,55.501,-269.999],[9E+09,9E+09,9E+09,9E+09,9E+09,9E+09]];

    CONST robtarget rA_t104 := [[2153.31,0.0367459,1279.08],[0.0943866,0.700781,0.700775,0.0943998],[0,0,-3,0],[9E+09,9E+09,9E+09,9E+09,9E+09,9E+09]];
    CONST robtarget rB_t104 := [[1089.62,-1227.12,-392.803],[0.443383,0.814828,0.331443,-0.172083],[-1,2,2,0],[9E+09,9E+09,9E+09,9E+09,9E+09,9E+09]];
    CONST robtarget rB_t104_c1 := [[1089.62,-1227.12,-392.803],[0.443383,0.814828,0.331443,-0.172083],[0,-4,-4,0],[9E+09,9E+09,9E+09,9E+09,9E+09,9E+09]];
    CONST jointtarget jA_t104 := [[0.00091901,13.5118,5.64439,0.000918909,55.501,-269.999],[9E+09,9E+09,9E+09,9E+09,9E+09,9E+09]];
    CONST jointtarget jB_t104 := [[-45.001,59.5019,28.5403,224.999,55.4021,224.999],[9E+09,9E+09,9E+09,9E+09,9E+09,9E+09]];
    CONST jointtarget jBseed_t104 := [[-45.001,59.5019,28.5403,224.999,55.4021,224.999],[9E+09,9E+09,9E+09,9E+09,9E+09,9E+09]];

    CONST robtarget rA_t107 := [[1115.03,-1254.27,3065.69],[0.5709,0.306712,0.0456818,-0.760207],[-1,2,1,0],[9E+09,9E+09,9E+09,9E+09,9E+09,9E+09]];
    CONST robtarget rB_t107 := [[-1653.03,-1752.06,2398.09],[0.670328,0.631027,-0.370983,0.121807],[-2,0,-3,0],[9E+09,9E+09,9E+09,9E+09,9E+09,9E+09]];
    CONST robtarget rB_t107_c5 := [[-1653.03,-1752.06,2398.09],[0.670328,0.631027,-0.370983,0.121807],[0,0,0,0],[9E+09,9E+09,9E+09,9E+09,9E+09,9E+09]];
    CONST jointtarget jA_t107 := [[-44.9996,18.5327,-61.373,225,56.4934,90.0004],[9E+09,9E+09,9E+09,9E+09,9E+09,9E+09]];
    CONST jointtarget jB_t107 := [[-134.999,31.7753,-54.7395,45.0008,36.3494,-269.999],[9E+09,9E+09,9E+09,9E+09,9E+09,9E+09]];
    CONST jointtarget jBseed_t107 := [[-134.999,31.7753,-54.7395,45.0008,36.3494,-269.999],[9E+09,9E+09,9E+09,9E+09,9E+09,9E+09]];

    CONST robtarget rA_t108 := [[-1653.03,-1752.06,2398.09],[0.670328,0.631027,-0.370983,0.121807],[-2,0,-3,0],[9E+09,9E+09,9E+09,9E+09,9E+09,9E+09]];
    CONST robtarget rB_t108 := [[-990.217,-861.447,2764.49],[0.155843,-0.330755,0.0341078,0.930135],[-2,2,-3,0],[9E+09,9E+09,9E+09,9E+09,9E+09,9E+09]];
    CONST robtarget rB_t108_c2 := [[-990.217,-861.447,2764.49],[0.155843,-0.330755,0.0341078,0.930135],[0,0,-4,0],[9E+09,9E+09,9E+09,9E+09,9E+09,9E+09]];
    CONST robtarget rB_t108_c3 := [[-990.217,-861.447,2764.49],[0.155843,-0.330755,0.0341078,0.930135],[0,4,-4,0],[9E+09,9E+09,9E+09,9E+09,9E+09,9E+09]];
    CONST jointtarget jA_t108 := [[-134.999,31.7753,-54.7395,45.0008,36.3494,-269.999],[9E+09,9E+09,9E+09,9E+09,9E+09,9E+09]];
    CONST jointtarget jB_t108 := [[-134.999,-17.6281,-10.0983,225.001,50.4618,-269.999],[9E+09,9E+09,9E+09,9E+09,9E+09,9E+09]];
    CONST jointtarget jBseed_t108 := [[-134.999,-17.6281,-10.0983,225.001,50.4617,-269.999],[9E+09,9E+09,9E+09,9E+09,9E+09,9E+09]];

    CONST robtarget rA_t109 := [[-990.217,-861.447,2764.49],[0.155843,-0.330755,0.0341078,0.930135],[-2,2,-3,0],[9E+09,9E+09,9E+09,9E+09,9E+09,9E+09]];
    CONST robtarget rB_t109 := [[-91.9691,-821.035,3431.33],[0.703236,-0.0740344,-0.325414,0.62776],[-2,-2,-2,0],[9E+09,9E+09,9E+09,9E+09,9E+09,9E+09]];
    CONST robtarget rB_t109_c6 := [[-91.9691,-821.035,3431.33],[0.703236,-0.0740344,-0.325414,0.62776],[0,4,0,0],[9E+09,9E+09,9E+09,9E+09,9E+09,9E+09]];
    CONST jointtarget jA_t109 := [[-134.999,-17.6281,-10.0983,225.001,50.4618,-269.999],[9E+09,9E+09,9E+09,9E+09,9E+09,9E+09]];
    CONST jointtarget jB_t109 := [[-90.0009,3.68605,-72.2953,-90.0009,33.4104,-90.001],[9E+09,9E+09,9E+09,9E+09,9E+09,9E+09]];
    CONST jointtarget jBseed_t109 := [[-90.0009,3.68603,-72.2953,-90.0009,33.4104,-90.0009],[9E+09,9E+09,9E+09,9E+09,9E+09,9E+09]];

    CONST robtarget rA_t110 := [[-91.9691,-821.035,3431.33],[0.703236,-0.0740344,-0.325414,0.62776],[-2,-2,-2,0],[9E+09,9E+09,9E+09,9E+09,9E+09,9E+09]];
    CONST robtarget rB_t110 := [[1351.39,1316.59,1723.27],[0.622769,-0.244608,0.716493,0.197393],[0,-2,0,0],[9E+09,9E+09,9E+09,9E+09,9E+09,9E+09]];
    CONST robtarget rB_t110_c2 := [[1351.39,1316.59,1723.27],[0.622769,-0.244608,0.716493,0.197393],[0,0,-4,0],[9E+09,9E+09,9E+09,9E+09,9E+09,9E+09]];
    CONST jointtarget jA_t110 := [[-90.0009,3.68605,-72.2953,-90.0009,33.4104,-90.001],[9E+09,9E+09,9E+09,9E+09,9E+09,9E+09]];
    CONST jointtarget jB_t110 := [[44.9998,-8.05139,16.5627,-90.0002,8.47072,89.9999],[9E+09,9E+09,9E+09,9E+09,9E+09,9E+09]];
    CONST jointtarget jBseed_t110 := [[44.9998,-8.0514,16.5627,-90.0002,8.47072,89.9998],[9E+09,9E+09,9E+09,9E+09,9E+09,9E+09]];

    CONST robtarget rA_t111 := [[1351.39,1316.59,1723.27],[0.622769,-0.244608,0.716493,0.197393],[0,-2,0,0],[9E+09,9E+09,9E+09,9E+09,9E+09,9E+09]];
    CONST robtarget rB_t111 := [[1481.28,1481.29,2644.16],[0.442284,-0.780241,4.35871E-7,-0.442276],[0,0,2,0],[9E+09,9E+09,9E+09,9E+09,9E+09,9E+09]];
    CONST robtarget rB_t111_c5 := [[1481.28,1481.29,2644.16],[0.442284,-0.780241,4.35871E-7,-0.442276],[0,0,0,0],[9E+09,9E+09,9E+09,9E+09,9E+09,9E+09]];
    CONST robtarget rB_t111_c8 := [[1481.28,1481.29,2644.16],[0.442284,-0.780241,4.35871E-7,-0.442276],[0,0,4,0],[9E+09,9E+09,9E+09,9E+09,9E+09,9E+09]];
    CONST jointtarget jA_t111 := [[44.9998,-8.05139,16.5627,-90.0002,8.47072,89.9999],[9E+09,9E+09,9E+09,9E+09,9E+09,9E+09]];
    CONST jointtarget jB_t111 := [[45.0003,19.7852,-50.2326,0.000301317,43.0128,225],[9E+09,9E+09,9E+09,9E+09,9E+09,9E+09]];
    CONST jointtarget jBseed_t111 := [[45.0003,19.7851,-50.2326,0.000301553,43.0128,225],[9E+09,9E+09,9E+09,9E+09,9E+09,9E+09]];

    CONST robtarget rA_t115 := [[2018.02,-2062.99,644.742],[0.307629,0.049721,0.850692,-0.423337],[-1,-1,0,0],[9E+09,9E+09,9E+09,9E+09,9E+09,9E+09]];
    CONST robtarget rB_t115 := [[2922.79,12.7726,1339.28],[0.463163,0.497358,0.53293,0.504083],[-1,1,-1,0],[9E+09,9E+09,9E+09,9E+09,9E+09,9E+09]];
    CONST robtarget rB_t115_c4 := [[2922.79,12.7726,1339.28],[0.463163,0.497358,0.53293,0.504083],[0,-4,0,0],[9E+09,9E+09,9E+09,9E+09,9E+09,9E+09]];
    CONST robtarget rB_t115_c5 := [[2922.79,12.7726,1339.28],[0.463163,0.497358,0.53293,0.504083],[0,0,0,0],[9E+09,9E+09,9E+09,9E+09,9E+09,9E+09]];
    CONST jointtarget jA_t115 := [[-44.9994,58.4655,-31.0303,-89.9994,10.9885,45.0006],[9E+09,9E+09,9E+09,9E+09,9E+09,9E+09]];
    CONST jointtarget jB_t115 := [[-0.000290098,51.4853,-43.4721,135,6.21662,-45.0003],[9E+09,9E+09,9E+09,9E+09,9E+09,9E+09]];
    CONST jointtarget jBseed_t115 := [[-0.000290078,51.4853,-43.4721,135,6.21662,-45.0003],[9E+09,9E+09,9E+09,9E+09,9E+09,9E+09]];

    CONST robtarget rA_t116 := [[2922.79,12.7726,1339.28],[0.463163,0.497358,0.53293,0.504083],[-1,1,-1,0],[9E+09,9E+09,9E+09,9E+09,9E+09,9E+09]];
    CONST robtarget rB_t116 := [[-0.00255183,1618.19,1254.41],[0.574215,-0.412649,-0.412648,-0.574213],[1,-2,0,0],[9E+09,9E+09,9E+09,9E+09,9E+09,9E+09]];
    CONST robtarget rB_t116_c2 := [[-0.00255183,1618.19,1254.41],[0.574215,-0.412649,-0.412648,-0.574213],[0,0,-4,0],[9E+09,9E+09,9E+09,9E+09,9E+09,9E+09]];
    CONST robtarget rB_t116_c5 := [[-0.00255183,1618.19,1254.41],[0.574215,-0.412649,-0.412648,-0.574213],[0,0,0,0],[9E+09,9E+09,9E+09,9E+09,9E+09,9E+09]];
    CONST jointtarget jA_t116 := [[-0.000290098,51.4853,-43.4721,135,6.21662,-45.0003],[9E+09,9E+09,9E+09,9E+09,9E+09,9E+09]];
    CONST jointtarget jB_t116 := [[90.0001,-16.7968,44.4496,-180,46.2484,9.77951E-5],[9E+09,9E+09,9E+09,9E+09,9E+09,9E+09]];
    CONST jointtarget jBseed_t116 := [[90.0001,-16.7968,44.4496,-180,46.2484,0.000101108],[9E+09,9E+09,9E+09,9E+09,9E+09,9E+09]];

    CONST robtarget rA_t117 := [[-0.00255183,1618.19,1254.41],[0.574215,-0.412649,-0.412648,-0.574213],[1,-2,0,0],[9E+09,9E+09,9E+09,9E+09,9E+09,9E+09]];
    CONST robtarget rB_t117 := [[1088.57,-1208.85,2577.78],[0.756806,0.311842,-0.224759,0.528661],[-1,-2,2,0],[9E+09,9E+09,9E+09,9E+09,9E+09,9E+09]];
    CONST robtarget rB_t117_c7 := [[1088.57,-1208.85,2577.78],[0.756806,0.311842,-0.224759,0.528661],[0,-4,4,0],[9E+09,9E+09,9E+09,9E+09,9E+09,9E+09]];
    CONST jointtarget jA_t117 := [[90.0001,-16.7968,44.4496,-180,46.2484,9.77951E-5],[9E+09,9E+09,9E+09,9E+09,9E+09,9E+09]];
    CONST jointtarget jB_t117 := [[-45.0003,-9.25626,-9.40794,-135,46.0653,270],[9E+09,9E+09,9E+09,9E+09,9E+09,9E+09]];
    CONST jointtarget jBseed_t117 := [[-45.0003,-9.25626,-9.40794,-135,46.0652,270],[9E+09,9E+09,9E+09,9E+09,9E+09,9E+09]];

    CONST robtarget rA_t119 := [[11.4262,2705.76,371.438],[0.135935,-0.358884,-0.827943,-0.408943],[1,3,-2,0],[9E+09,9E+09,9E+09,9E+09,9E+09,9E+09]];
    CONST robtarget rB_t119 := [[1236.14,-1341.56,-176.736],[0.406944,0.85015,0.322838,-0.086124],[-1,2,-2,0],[9E+09,9E+09,9E+09,9E+09,9E+09,9E+09]];
    CONST robtarget rB_t119_c1 := [[1236.14,-1341.56,-176.736],[0.406944,0.85015,0.322838,-0.086124],[0,-4,-4,0],[9E+09,9E+09,9E+09,9E+09,9E+09,9E+09]];
    CONST jointtarget jA_t119 := [[90.0001,56.0118,-16.9579,270,3.92407,-135],[9E+09,9E+09,9E+09,9E+09,9E+09,9E+09]];
    CONST jointtarget jB_t119 := [[-45.0001,49.7201,27.1517,225,39.14,-135],[9E+09,9E+09,9E+09,9E+09,9E+09,9E+09]];
    CONST jointtarget jBseed_t119 := [[-45.0001,49.7201,27.1517,225,39.14,-135],[9E+09,9E+09,9E+09,9E+09,9E+09,9E+09]];

    CONST robtarget rA_t122 := [[1179.46,1260.01,1671.71],[0.640292,-0.73583,0.183252,-0.122465],[0,0,-3,0],[9E+09,9E+09,9E+09,9E+09,9E+09,9E+09]];
    CONST robtarget rB_t122 := [[788.046,-907.763,3177.9],[0.9238,0.182587,-0.200201,0.270509],[-1,-2,-2,0],[9E+09,9E+09,9E+09,9E+09,9E+09,9E+09]];
    CONST robtarget rB_t122_c1 := [[788.046,-907.763,3177.9],[0.9238,0.182587,-0.200201,0.270509],[0,-4,-4,0],[9E+09,9E+09,9E+09,9E+09,9E+09,9E+09]];
    CONST robtarget rB_t122_c2 := [[788.046,-907.763,3177.9],[0.9238,0.182587,-0.200201,0.270509],[0,0,-4,0],[9E+09,9E+09,9E+09,9E+09,9E+09,9E+09]];
    CONST jointtarget jA_t122 := [[44.9993,-16.046,25.2315,89.9993,19.95,-180.001],[9E+09,9E+09,9E+09,9E+09,9E+09,9E+09]];
    CONST jointtarget jB_t122 := [[-45.0006,-3.98999,-41.7661,-135.001,45.7888,-135.001],[9E+09,9E+09,9E+09,9E+09,9E+09,9E+09]];
    CONST jointtarget jBseed_t122 := [[-45.0006,-3.98999,-41.7661,-135.001,45.7888,-135.001],[9E+09,9E+09,9E+09,9E+09,9E+09,9E+09]];

    CONST robtarget rA_t124 := [[2444.64,27.9798,6.20578],[0.0799213,-0.946671,-0.0262629,-0.311027],[-1,0,-4,0],[9E+09,9E+09,9E+09,9E+09,9E+09,9E+09]];
    CONST robtarget rB_t124 := [[965.012,93.2527,2528.1],[0.480133,0.162498,0.519118,0.688174],[-1,-4,-5,0],[9E+09,9E+09,9E+09,9E+09,9E+09,9E+09]];
    CONST robtarget rB_t124_c5 := [[965.012,93.2527,2528.1],[0.480133,0.162498,0.519118,0.688174],[0,0,0,0],[9E+09,9E+09,9E+09,9E+09,9E+09,9E+09]];
    CONST jointtarget jA_t124 := [[-0.000453385,57.843,-4.21857,89.9995,9.65178,-270],[9E+09,9E+09,9E+09,9E+09,9E+09,9E+09]];
    CONST jointtarget jB_t124 := [[-0.000517769,-40.2936,10.8139,-270.001,33.9488,-360.001],[9E+09,9E+09,9E+09,9E+09,9E+09,9E+09]];
    CONST jointtarget jBseed_t124 := [[-0.000517563,-40.2936,10.8139,-270.001,33.9488,-360.001],[9E+09,9E+09,9E+09,9E+09,9E+09,9E+09]];

    CONST robtarget rA_t126 := [[0.044724,2908.86,1076.14],[0.542717,-0.453293,0.453283,0.542696],[0,-3,1,0],[9E+09,9E+09,9E+09,9E+09,9E+09,9E+09]];
    CONST robtarget rB_t126 := [[-1429.64,1300.22,965.752],[0.304325,0.144439,-0.938743,0.0726961],[1,0,1,0],[9E+09,9E+09,9E+09,9E+09,9E+09,9E+09]];
    CONST robtarget rB_t126_c5 := [[-1429.64,1300.22,965.752],[0.304325,0.144439,-0.938743,0.0726961],[0,0,0,0],[9E+09,9E+09,9E+09,9E+09,9E+09,9E+09]];
    CONST jointtarget jA_t126 := [[89.9991,52.888,-34.4621,-180.001,28.6862,179.999],[9E+09,9E+09,9E+09,9E+09,9E+09,9E+09]];
    CONST jointtarget jB_t126 := [[135.001,8.5348,24.565,45.0009,50.7822,90.0009],[9E+09,9E+09,9E+09,9E+09,9E+09,9E+09]];
    CONST jointtarget jBseed_t126 := [[135.001,8.53481,24.565,45.0009,50.7822,90.0009],[9E+09,9E+09,9E+09,9E+09,9E+09,9E+09]];

    CONST robtarget rA_t129 := [[-1497.57,-1497.53,2172.3],[0.352555,0.353726,-0.853967,0.146023],[-2,-1,1,0],[9E+09,9E+09,9E+09,9E+09,9E+09,9E+09]];
    CONST robtarget rB_t129 := [[-1827.84,-1827.87,2250.12],[0.346324,0.393108,0.162827,-0.83607],[-2,-2,2,0],[9E+09,9E+09,9E+09,9E+09,9E+09,9E+09]];
    CONST robtarget rB_t129_c4 := [[-1827.84,-1827.87,2250.12],[0.346324,0.393108,0.162827,-0.83607],[0,-4,0,0],[9E+09,9E+09,9E+09,9E+09,9E+09,9E+09]];
    CONST robtarget rB_t129_c5 := [[-1827.84,-1827.87,2250.12],[0.346324,0.393108,0.162827,-0.83607],[0,0,0,0],[9E+09,9E+09,9E+09,9E+09,9E+09,9E+09]];
    CONST jointtarget jA_t129 := [[-135.001,10.7541,-22.8693,-0.000633003,57.2497,179.999],[9E+09,9E+09,9E+09,9E+09,9E+09,9E+09]];
    CONST jointtarget jB_t129 := [[-134.999,38.2611,-53.2795,-179.999,24.6175,180.001],[9E+09,9E+09,9E+09,9E+09,9E+09,9E+09]];
    CONST jointtarget jBseed_t129 := [[-134.999,38.2611,-53.2795,-179.999,24.6175,180.001],[9E+09,9E+09,9E+09,9E+09,9E+09,9E+09]];

    CONST robtarget rA_t131 := [[-32.8128,-2624.37,515.297],[0.44033,0.803566,0.286796,-0.279535],[-1,-2,2,0],[9E+09,9E+09,9E+09,9E+09,9E+09,9E+09]];
    CONST robtarget rB_t131 := [[1626.2,-1630.26,2180.78],[0.28541,-0.242978,0.60349,-0.703778],[-1,2,0,0],[9E+09,9E+09,9E+09,9E+09,9E+09,9E+09]];
    CONST robtarget rB_t131_c4 := [[1626.2,-1630.26,2180.78],[0.28541,-0.242978,0.60349,-0.703778],[0,-4,0,0],[9E+09,9E+09,9E+09,9E+09,9E+09,9E+09]];
    CONST jointtarget jA_t131 := [[-89.9992,48.204,-8.91995,-134.999,16.1504,180.001],[9E+09,9E+09,9E+09,9E+09,9E+09,9E+09]];
    CONST jointtarget jB_t131 := [[-45.0002,16.1742,-24.0239,225,1.38981,44.9996],[9E+09,9E+09,9E+09,9E+09,9E+09,9E+09]];
    CONST jointtarget jBseed_t131 := [[-45.0002,16.1742,-24.0239,225,1.38981,44.9998],[9E+09,9E+09,9E+09,9E+09,9E+09,9E+09]];

    CONST robtarget rA_t133 := [[1662.3,-0.0172653,709.662],[0.109355,-0.379997,0.917383,-0.0453009],[-1,-1,-1,0],[9E+09,9E+09,9E+09,9E+09,9E+09,9E+09]];
    CONST robtarget rB_t133 := [[-0.0268639,2431.67,974.659],[0.464529,-0.533107,0.533114,0.464542],[1,2,-2,0],[9E+09,9E+09,9E+09,9E+09,9E+09,9E+09]];
    CONST robtarget rB_t133_c2 := [[-0.0268639,2431.67,974.659],[0.464529,-0.533107,0.533114,0.464542],[0,0,-4,0],[9E+09,9E+09,9E+09,9E+09,9E+09,9E+09]];
    CONST jointtarget jA_t133 := [[-0.000564186,2.08564,41.2836,-0.000564374,33.0351,-45.0006],[9E+09,9E+09,9E+09,9E+09,9E+09,9E+09]];
    CONST jointtarget jB_t133 := [[90.0006,28.3328,3.98602,180.001,24.4545,-179.999],[9E+09,9E+09,9E+09,9E+09,9E+09,9E+09]];
    CONST jointtarget jBseed_t133 := [[90.0006,28.3328,3.98602,180.001,24.4545,-179.999],[9E+09,9E+09,9E+09,9E+09,9E+09,9E+09]];

    CONST robtarget rA_t134 := [[-0.0268639,2431.67,974.659],[0.464529,-0.533107,0.533114,0.464542],[1,2,-2,0],[9E+09,9E+09,9E+09,9E+09,9E+09,9E+09]];
    CONST robtarget rB_t134 := [[-858.78,865.991,3043.68],[0.916715,-0.292126,-0.2725,-0.00630857],[1,-2,-1,0],[9E+09,9E+09,9E+09,9E+09,9E+09,9E+09]];
    CONST robtarget rB_t134_c2 := [[-858.78,865.991,3043.68],[0.916715,-0.292126,-0.2725,-0.00630857],[0,0,-4,0],[9E+09,9E+09,9E+09,9E+09,9E+09,9E+09]];
    CONST robtarget rB_t134_c5 := [[-858.78,865.991,3043.68],[0.916715,-0.292126,-0.2725,-0.00630857],[0,0,0,0],[9E+09,9E+09,9E+09,9E+09,9E+09,9E+09]];
    CONST jointtarget jA_t134 := [[90.0006,28.3328,3.98602,180.001,24.4545,-179.999],[9E+09,9E+09,9E+09,9E+09,9E+09,9E+09]];
    CONST jointtarget jB_t134 := [[135,-13.1895,-27.9952,-135,2.47017,-0.000378917],[9E+09,9E+09,9E+09,9E+09,9E+09,9E+09]];
    CONST jointtarget jBseed_t134 := [[135,-13.1895,-27.9952,-135,2.47017,-0.000435102],[9E+09,9E+09,9E+09,9E+09,9E+09,9E+09]];

    CONST robtarget rA_t142 := [[473.483,0.00208691,3479.51],[0.923192,-0.0147901,0.0357082,-0.382391],[0,-2,-3,0],[9E+09,9E+09,9E+09,9E+09,9E+09,9E+09]];
    CONST robtarget rB_t142 := [[1417.42,1360.7,2365.48],[0.0771357,0.440595,0.307005,0.840044],[0,-2,3,0],[9E+09,9E+09,9E+09,9E+09,9E+09,9E+09]];
    CONST robtarget rB_t142_c5 := [[1417.42,1360.7,2365.48],[0.0771357,0.440595,0.307005,0.840044],[0,0,0,0],[9E+09,9E+09,9E+09,9E+09,9E+09,9E+09]];
    CONST jointtarget jA_t142 := [[0.00027492,-7.69249,-64.2137,-180,13.6637,-225],[9E+09,9E+09,9E+09,9E+09,9E+09,9E+09]];
    CONST jointtarget jB_t142 := [[45.0006,1.13346,-12.6533,-134.999,19.8639,270.001],[9E+09,9E+09,9E+09,9E+09,9E+09,9E+09]];
    CONST jointtarget jBseed_t142 := [[45.0006,1.13346,-12.6533,-134.999,19.8639,270.001],[9E+09,9E+09,9E+09,9E+09,9E+09,9E+09]];

    CONST robtarget rA_t143 := [[1417.42,1360.7,2365.48],[0.0771357,0.440595,0.307005,0.840044],[0,-2,3,0],[9E+09,9E+09,9E+09,9E+09,9E+09,9E+09]];
    CONST robtarget rB_t143 := [[49.5001,2643.04,881.323],[0.618466,-0.771015,0.0756653,-0.13157],[1,-2,-4,0],[9E+09,9E+09,9E+09,9E+09,9E+09,9E+09]];
    CONST robtarget rB_t143_c5 := [[49.5001,2643.04,881.323],[0.618466,-0.771015,0.0756653,-0.13157],[0,0,0,0],[9E+09,9E+09,9E+09,9E+09,9E+09,9E+09]];
    CONST jointtarget jA_t143 := [[45.0006,1.13346,-12.6533,-134.999,19.8639,270.001],[9E+09,9E+09,9E+09,9E+09,9E+09,9E+09]];
    CONST jointtarget jB_t143 := [[90.0003,40.6085,-10.4117,-135,24.7896,-315],[9E+09,9E+09,9E+09,9E+09,9E+09,9E+09]];
    CONST jointtarget jBseed_t143 := [[90.0003,40.6085,-10.4117,-135,24.7896,-315],[9E+09,9E+09,9E+09,9E+09,9E+09,9E+09]];

    CONST robtarget rA_t149 := [[848.546,879.856,1952.09],[0.264086,0.18407,0.575738,0.7516],[0,1,3,0],[9E+09,9E+09,9E+09,9E+09,9E+09,9E+09]];
    CONST robtarget rB_t149 := [[0.0017069,512.734,3460.73],[0.698154,0.112191,-0.112192,0.698146],[0,-3,-3,0],[9E+09,9E+09,9E+09,9E+09,9E+09,9E+09]];
    CONST robtarget rB_t149_c5 := [[0.0017069,512.734,3460.73],[0.698154,0.112191,-0.112192,0.698146],[0,0,0,0],[9E+09,9E+09,9E+09,9E+09,9E+09,9E+09]];
    CONST jointtarget jA_t149 := [[45.0002,-42.8132,34.7334,135,10.8036,315],[9E+09,9E+09,9E+09,9E+09,9E+09,9E+09]];
    CONST jointtarget jB_t149 := [[89.9998,-5.92366,-63.3488,-180,38.9862,-180],[9E+09,9E+09,9E+09,9E+09,9E+09,9E+09]];
    CONST jointtarget jBseed_t149 := [[89.9998,-5.92365,-63.3488,-180,38.9862,-180],[9E+09,9E+09,9E+09,9E+09,9E+09,9E+09]];

    CONST robtarget rA_t152 := [[1811.76,-1811.81,1422.18],[0.52547,-6.42825E-6,0.669135,-0.52549],[-1,-3,1,0],[9E+09,9E+09,9E+09,9E+09,9E+09,9E+09]];
    CONST robtarget rB_t152 := [[-67.2679,-2277.56,1614.19],[0.323488,0.204447,-0.850609,0.360585],[-1,-1,3,0],[9E+09,9E+09,9E+09,9E+09,9E+09,9E+09]];
    CONST robtarget rB_t152_c8 := [[-67.2679,-2277.56,1614.19],[0.323488,0.204447,-0.850609,0.360585],[0,0,4,0],[9E+09,9E+09,9E+09,9E+09,9E+09,9E+09]];
    CONST jointtarget jA_t152 := [[-45.0008,28.5781,-12.0383,-180.001,22.5391,134.999],[9E+09,9E+09,9E+09,9E+09,9E+09,9E+09]];
    CONST jointtarget jB_t152 := [[-89.9996,14.138,-4.81765,-44.9996,34.7343,270],[9E+09,9E+09,9E+09,9E+09,9E+09,9E+09]];
    CONST jointtarget jBseed_t152 := [[-89.9996,14.138,-4.81765,-44.9996,34.7343,270],[9E+09,9E+09,9E+09,9E+09,9E+09,9E+09]];

    CONST robtarget rA_t153 := [[-67.2679,-2277.56,1614.19],[0.323488,0.204447,-0.850609,0.360585],[-1,-1,3,0],[9E+09,9E+09,9E+09,9E+09,9E+09,9E+09]];
    CONST robtarget rB_t153 := [[1879.57,-1918.72,2009.23],[0.758875,0.5015,0.411947,-0.053901],[-1,2,1,0],[9E+09,9E+09,9E+09,9E+09,9E+09,9E+09]];
    CONST robtarget rB_t153_c5 := [[1879.57,-1918.72,2009.23],[0.758875,0.5015,0.411947,-0.053901],[0,0,0,0],[9E+09,9E+09,9E+09,9E+09,9E+09,9E+09]];
    CONST jointtarget jA_t153 := [[-89.9996,14.138,-4.81765,-44.9996,34.7343,270],[9E+09,9E+09,9E+09,9E+09,9E+09,9E+09]];
    CONST jointtarget jB_t153 := [[-45.0001,39.1803,-48.3758,270,9.54008,135],[9E+09,9E+09,9E+09,9E+09,9E+09,9E+09]];
    CONST jointtarget jBseed_t153 := [[-45.0001,39.1803,-48.3758,270,9.54009,135],[9E+09,9E+09,9E+09,9E+09,9E+09,9E+09]];

    CONST robtarget rA_t154 := [[1879.57,-1918.72,2009.23],[0.758875,0.5015,0.411947,-0.053901],[-1,2,1,0],[9E+09,9E+09,9E+09,9E+09,9E+09,9E+09]];
    CONST robtarget rB_t154 := [[1780.64,1974.64,1682.3],[0.612395,-0.679367,0.226242,0.335034],[0,-4,-2,0],[9E+09,9E+09,9E+09,9E+09,9E+09,9E+09]];
    CONST robtarget rB_t154_c5 := [[1780.64,1974.64,1682.3],[0.612395,-0.679367,0.226242,0.335034],[0,0,0,0],[9E+09,9E+09,9E+09,9E+09,9E+09,9E+09]];
    CONST jointtarget jA_t154 := [[-45.0001,39.1803,-48.3758,270,9.54008,135],[9E+09,9E+09,9E+09,9E+09,9E+09,9E+09]];
    CONST jointtarget jB_t154 := [[44.9997,37.73,-35.1723,-270,55.2373,-135],[9E+09,9E+09,9E+09,9E+09,9E+09,9E+09]];
    CONST jointtarget jBseed_t154 := [[44.9997,37.73,-35.1723,-270,55.2373,-135],[9E+09,9E+09,9E+09,9E+09,9E+09,9E+09]];

    CONST robtarget rA_t157 := [[527.04,462.715,2891.3],[0.416445,0.218217,0.193782,0.861048],[0,2,-2,0],[9E+09,9E+09,9E+09,9E+09,9E+09,9E+09]];
    CONST robtarget rB_t157 := [[0.0173601,-2251.83,1472.37],[0.678452,0.627107,0.259752,-0.281016],[-1,-2,-2,0],[9E+09,9E+09,9E+09,9E+09,9E+09,9E+09]];
    CONST robtarget rB_t157_c8 := [[0.0173601,-2251.83,1472.37],[0.678452,0.627107,0.259752,-0.281016],[0,0,4,0],[9E+09,9E+09,9E+09,9E+09,9E+09,9E+09]];
    CONST jointtarget jA_t157 := [[45.0005,-38.305,-4.82162,225.001,22.6582,-134.999],[9E+09,9E+09,9E+09,9E+09,9E+09,9E+09]];
    CONST jointtarget jB_t157 := [[-89.9995,12.1238,6.54104,-180,23.169,-135],[9E+09,9E+09,9E+09,9E+09,9E+09,9E+09]];
    CONST jointtarget jBseed_t157 := [[-89.9995,12.1238,6.54103,-180,23.169,-135],[9E+09,9E+09,9E+09,9E+09,9E+09,9E+09]];

    CONST robtarget rA_t159 := [[-1885.86,1966.19,1817.66],[0.338933,-0.12966,-0.78238,-0.506157],[1,-1,-3,0],[9E+09,9E+09,9E+09,9E+09,9E+09,9E+09]];
    CONST robtarget rB_t159 := [[1784.99,1852.33,343.96],[0.319104,-0.762341,-0.3761,-0.418995],[0,1,0,0],[9E+09,9E+09,9E+09,9E+09,9E+09,9E+09]];
    CONST robtarget rB_t159_c4 := [[1784.99,1852.33,343.96],[0.319104,-0.762341,-0.3761,-0.418995],[0,-4,0,0],[9E+09,9E+09,9E+09,9E+09,9E+09,9E+09]];
    CONST jointtarget jA_t159 := [[134.999,40.6928,-45.9716,-45.0005,28.7375,-180.001],[9E+09,9E+09,9E+09,9E+09,9E+09,9E+09]];
    CONST jointtarget jB_t159 := [[45.0008,51.2912,-6.32526,135.001,23.7587,45.0008],[9E+09,9E+09,9E+09,9E+09,9E+09,9E+09]];
    CONST jointtarget jBseed_t159 := [[45.0008,51.2912,-6.32526,135.001,23.7587,45.0008],[9E+09,9E+09,9E+09,9E+09,9E+09,9E+09]];

    CONST robtarget rA_t163 := [[38.7719,-1203.89,3366.29],[0.984467,0.130213,0.114103,0.0291624],[-2,1,3,0],[9E+09,9E+09,9E+09,9E+09,9E+09,9E+09]];
    CONST robtarget rB_t163 := [[-7.02831,1267.92,3085.7],[0.653554,-0.269952,-0.297191,-0.641616],[1,1,1,0],[9E+09,9E+09,9E+09,9E+09,9E+09,9E+09]];
    CONST robtarget rB_t163_c5 := [[-7.02831,1267.92,3085.7],[0.653554,-0.269952,-0.297191,-0.641616],[0,0,0,0],[9E+09,9E+09,9E+09,9E+09,9E+09,9E+09]];
    CONST jointtarget jA_t163 := [[-90.0007,14.1966,-75.505,134.999,19.1754,314.999],[9E+09,9E+09,9E+09,9E+09,9E+09,9E+09]];
    CONST jointtarget jB_t163 := [[90.0003,-9.05484,-33.6488,90.0002,2.40974,90.0004],[9E+09,9E+09,9E+09,9E+09,9E+09,9E+09]];
    CONST jointtarget jBseed_t163 := [[90.0003,-9.05484,-33.6488,90.0003,2.40974,90.0003],[9E+09,9E+09,9E+09,9E+09,9E+09,9E+09]];

    CONST robtarget rA_t165 := [[-1376.09,-1480.75,2644.27],[0.738677,0.332889,0.194729,-0.552831],[-2,1,-2,0],[9E+09,9E+09,9E+09,9E+09,9E+09,9E+09]];
    CONST robtarget rB_t165 := [[-47.1012,-2479.06,2130.99],[0.229668,0.306112,0.456394,-0.803276],[-1,2,1,0],[9E+09,9E+09,9E+09,9E+09,9E+09,9E+09]];
    CONST robtarget rB_t165_c3 := [[-47.1012,-2479.06,2130.99],[0.229668,0.306112,0.456394,-0.803276],[0,4,-4,0],[9E+09,9E+09,9E+09,9E+09,9E+09,9E+09]];
    CONST robtarget rB_t165_c6 := [[-47.1012,-2479.06,2130.99],[0.229668,0.306112,0.456394,-0.803276],[0,4,0,0],[9E+09,9E+09,9E+09,9E+09,9E+09,9E+09]];
    CONST jointtarget jA_t165 := [[-135,12.7317,-34.7041,135,38.8086,-90.0001],[9E+09,9E+09,9E+09,9E+09,9E+09,9E+09]];
    CONST jointtarget jB_t165 := [[-89.9996,26.7104,-33.986,225,23.517,90.0004],[9E+09,9E+09,9E+09,9E+09,9E+09,9E+09]];
    CONST jointtarget jBseed_t165 := [[-89.9996,26.7104,-33.986,225,23.517,90.0004],[9E+09,9E+09,9E+09,9E+09,9E+09,9E+09]];

    CONST robtarget rA_t166 := [[-47.1012,-2479.06,2130.99],[0.229668,0.306112,0.456394,-0.803276],[-1,2,1,0],[9E+09,9E+09,9E+09,9E+09,9E+09,9E+09]];
    CONST robtarget rB_t166 := [[1385.94,1477.41,2037.54],[0.0875148,0.170606,0.797563,0.571951],[0,0,0,0],[9E+09,9E+09,9E+09,9E+09,9E+09,9E+09]];
    CONST robtarget rB_t166_c5 := [[1385.94,1477.41,2037.54],[0.0875148,0.170606,0.797563,0.571951],[0,0,0,0],[9E+09,9E+09,9E+09,9E+09,9E+09,9E+09]];
    CONST jointtarget jA_t166 := [[-89.9996,26.7104,-33.986,225,23.517,90.0004],[9E+09,9E+09,9E+09,9E+09,9E+09,9E+09]];
    CONST jointtarget jB_t166 := [[44.9999,1.55096,-5.38896,44.9999,33.2108,44.9999],[9E+09,9E+09,9E+09,9E+09,9E+09,9E+09]];
    CONST jointtarget jBseed_t166 := [[44.9999,1.55095,-5.38895,44.9999,33.2108,44.9999],[9E+09,9E+09,9E+09,9E+09,9E+09,9E+09]];

    CONST robtarget rA_t167 := [[1385.94,1477.41,2037.54],[0.0875148,0.170606,0.797563,0.571951],[0,0,0,0],[9E+09,9E+09,9E+09,9E+09,9E+09,9E+09]];
    CONST robtarget rB_t167 := [[-14.2891,2521.58,1560.78],[0.60744,-0.793202,-0.0275883,0.0329587],[0,0,2,0],[9E+09,9E+09,9E+09,9E+09,9E+09,9E+09]];
    CONST robtarget rB_t167_c2 := [[-14.2891,2521.58,1560.78],[0.60744,-0.793202,-0.0275883,0.0329587],[0,0,-4,0],[9E+09,9E+09,9E+09,9E+09,9E+09,9E+09]];
    CONST robtarget rB_t167_c5 := [[-14.2891,2521.58,1560.78],[0.60744,-0.793202,-0.0275883,0.0329587],[0,0,0,0],[9E+09,9E+09,9E+09,9E+09,9E+09,9E+09]];
    CONST jointtarget jA_t167 := [[44.9999,1.55096,-5.38896,44.9999,33.2108,44.9999],[9E+09,9E+09,9E+09,9E+09,9E+09,9E+09]];
    CONST jointtarget jB_t167 := [[89.999,25.5165,-15.3392,44.999,6.97104,224.999],[9E+09,9E+09,9E+09,9E+09,9E+09,9E+09]];
    CONST jointtarget jBseed_t167 := [[89.999,25.5165,-15.3392,44.999,6.97104,224.999],[9E+09,9E+09,9E+09,9E+09,9E+09,9E+09]];

    CONST robtarget rA_t170 := [[1102.23,-1245.72,3078.14],[0.917545,0.138376,-0.291101,0.232859],[-1,-2,-2,0],[9E+09,9E+09,9E+09,9E+09,9E+09,9E+09]];
    CONST robtarget rB_t170 := [[1183.72,-1023.77,598.794],[0.0275546,-0.880476,-0.118757,-0.458148],[-1,1,0,0],[9E+09,9E+09,9E+09,9E+09,9E+09,9E+09]];
    CONST robtarget rB_t170_c4 := [[1183.72,-1023.77,598.794],[0.0275546,-0.880476,-0.118757,-0.458148],[0,-4,0,0],[9E+09,9E+09,9E+09,9E+09,9E+09,9E+09]];
    CONST jointtarget jA_t170 := [[-44.9999,19.8108,-64.0034,-135,59.2328,-135],[9E+09,9E+09,9E+09,9E+09,9E+09,9E+09]];
    CONST jointtarget jB_t170 := [[-44.9991,2.64962,49.1986,90.0008,42.6173,45.0009],[9E+09,9E+09,9E+09,9E+09,9E+09,9E+09]];
    CONST jointtarget jBseed_t170 := [[-44.9991,2.64962,49.1986,90.0009,42.6173,45.0009],[9E+09,9E+09,9E+09,9E+09,9E+09,9E+09]];

    CONST robtarget rA_t171 := [[1183.72,-1023.77,598.794],[0.0275546,-0.880476,-0.118757,-0.458148],[-1,1,0,0],[9E+09,9E+09,9E+09,9E+09,9E+09,9E+09]];
    CONST robtarget rB_t171 := [[1631.88,-1711.11,435.706],[0.407611,0.379998,0.755878,-0.343662],[-1,-2,-3,0],[9E+09,9E+09,9E+09,9E+09,9E+09,9E+09]];
    CONST robtarget rB_t171_c4 := [[1631.88,-1711.11,435.706],[0.407611,0.379998,0.755878,-0.343662],[0,-4,0,0],[9E+09,9E+09,9E+09,9E+09,9E+09,9E+09]];
    CONST robtarget rB_t171_c5 := [[1631.88,-1711.11,435.706],[0.407611,0.379998,0.755878,-0.343662],[0,0,0,0],[9E+09,9E+09,9E+09,9E+09,9E+09,9E+09]];
    CONST jointtarget jA_t171 := [[-44.9991,2.64962,49.1986,90.0008,42.6173,45.0009],[9E+09,9E+09,9E+09,9E+09,9E+09,9E+09]];
    CONST jointtarget jB_t171 := [[-45.0005,40.1324,7.9812,-135,28.3126,-225],[9E+09,9E+09,9E+09,9E+09,9E+09,9E+09]];
    CONST jointtarget jBseed_t171 := [[-45.0005,40.1324,7.9812,-135,28.3126,-225],[9E+09,9E+09,9E+09,9E+09,9E+09,9E+09]];

    CONST robtarget rA_t174 := [[1613.53,90.3056,2898.4],[0.392626,0.279976,0.659378,0.576784],[-1,0,-4,0],[9E+09,9E+09,9E+09,9E+09,9E+09,9E+09]];
    CONST robtarget rB_t174 := [[37.749,-71.2403,3117.89],[0.326606,0.0916654,0.199448,-0.919318],[0,2,-4,0],[9E+09,9E+09,9E+09,9E+09,9E+09,9E+09]];
    CONST robtarget rB_t174_c3 := [[37.749,-71.2403,3117.89],[0.326606,0.0916654,0.199448,-0.919318],[0,4,-4,0],[9E+09,9E+09,9E+09,9E+09,9E+09,9E+09]];
    CONST jointtarget jA_t174 := [[-0.000215401,3.12203,-41.3376,44.9998,49.8886,-315],[9E+09,9E+09,9E+09,9E+09,9E+09,9E+09]];
    CONST jointtarget jB_t174 := [[0.000285623,-43.2344,-21.0483,225,37.1056,-360],[9E+09,9E+09,9E+09,9E+09,9E+09,9E+09]];
    CONST jointtarget jBseed_t174 := [[0.000283609,-43.2344,-21.0483,225,37.1056,-360],[9E+09,9E+09,9E+09,9E+09,9E+09,9E+09]];

    CONST robtarget rA_t177 := [[-950.268,-954.595,-396.793],[0.0174734,0.382765,0.923497,0.0183916],[-2,-3,-2,0],[9E+09,9E+09,9E+09,9E+09,9E+09,9E+09]];
    CONST robtarget rB_t177 := [[-0.00968228,-1814.57,2499.09],[0.904061,0.19032,0.0788361,-0.374482],[-2,1,-2,0],[9E+09,9E+09,9E+09,9E+09,9E+09,9E+09]];
    CONST robtarget rB_t177_c1 := [[-0.00968228,-1814.57,2499.09],[0.904061,0.19032,0.0788361,-0.374482],[0,-4,-4,0],[9E+09,9E+09,9E+09,9E+09,9E+09,9E+09]];
    CONST jointtarget jA_t177 := [[-134.999,54.1954,38.5183,-269.999,1.04373,-179.999],[9E+09,9E+09,9E+09,9E+09,9E+09,9E+09]];
    CONST jointtarget jB_t177 := [[-90.0003,-1.55827,-11.9788,180,52.6866,-135],[9E+09,9E+09,9E+09,9E+09,9E+09,9E+09]];
    CONST jointtarget jBseed_t177 := [[-90.0003,-1.55827,-11.9788,180,52.6865,-135],[9E+09,9E+09,9E+09,9E+09,9E+09,9E+09]];

    CONST robtarget rA_t183 := [[-854.508,989.938,1722.61],[0.102876,-0.0348942,-0.486379,-0.866968],[1,2,-2,0],[9E+09,9E+09,9E+09,9E+09,9E+09,9E+09]];
    CONST robtarget rB_t183 := [[-27.8139,2850.55,1136.14],[0.313825,-0.240648,-0.711151,-0.581263],[0,1,-5,0],[9E+09,9E+09,9E+09,9E+09,9E+09,9E+09]];
    CONST robtarget rB_t183_c2 := [[-27.8139,2850.55,1136.14],[0.313825,-0.240648,-0.711151,-0.581263],[0,0,-4,0],[9E+09,9E+09,9E+09,9E+09,9E+09,9E+09]];
    CONST robtarget rB_t183_c5 := [[-27.8139,2850.55,1136.14],[0.313825,-0.240648,-0.711151,-0.581263],[0,0,0,0],[9E+09,9E+09,9E+09,9E+09,9E+09,9E+09]];
    CONST jointtarget jA_t183 := [[135,-37.3492,41.97,225,54.1899,-135],[9E+09,9E+09,9E+09,9E+09,9E+09,9E+09]];
    CONST jointtarget jB_t183 := [[89.9998,47.7901,-30.6455,135,13.6271,-360],[9E+09,9E+09,9E+09,9E+09,9E+09,9E+09]];
    CONST jointtarget jBseed_t183 := [[89.9998,47.7902,-30.6455,135,13.6271,-360],[9E+09,9E+09,9E+09,9E+09,9E+09,9E+09]];

    CONST robtarget rA_t187 := [[52.7694,2089.12,1907.93],[0.115773,0.110421,0.714269,0.681339],[0,-2,1,0],[9E+09,9E+09,9E+09,9E+09,9E+09,9E+09]];
    CONST robtarget rB_t187 := [[-105.554,-98.573,3049.82],[0.916803,0.216637,-0.326479,-0.0771468],[-2,-2,-3,0],[9E+09,9E+09,9E+09,9E+09,9E+09,9E+09]];
    CONST robtarget rB_t187_c6 := [[-105.554,-98.573,3049.82],[0.916803,0.216637,-0.326479,-0.0771468],[0,4,0,0],[9E+09,9E+09,9E+09,9E+09,9E+09,9E+09]];
    CONST jointtarget jA_t187 := [[89.9994,2.84738,-0.144049,-90.0006,18.4118,179.999],[9E+09,9E+09,9E+09,9E+09,9E+09,9E+09]];
    CONST jointtarget jB_t187 := [[-90,-45.0874,-18.3227,-90,39.2022,-180],[9E+09,9E+09,9E+09,9E+09,9E+09,9E+09]];
    CONST jointtarget jBseed_t187 := [[-90,-45.0874,-18.3227,-90,39.2022,-180],[9E+09,9E+09,9E+09,9E+09,9E+09,9E+09]];

    CONST robtarget rA_t188 := [[-105.554,-98.573,3049.82],[0.916803,0.216637,-0.326479,-0.0771468],[-2,-2,-3,0],[9E+09,9E+09,9E+09,9E+09,9E+09,9E+09]];
    CONST robtarget rB_t188 := [[1056.67,1056.64,3185.67],[0.354669,-0.34688,-0.143685,-0.856294],[0,-1,1,0],[9E+09,9E+09,9E+09,9E+09,9E+09,9E+09]];
    CONST robtarget rB_t188_c2 := [[1056.67,1056.64,3185.67],[0.354669,-0.34688,-0.143685,-0.856294],[0,0,-4,0],[9E+09,9E+09,9E+09,9E+09,9E+09,9E+09]];
    CONST jointtarget jA_t188 := [[-90,-45.0874,-18.3227,-90,39.2022,-180],[9E+09,9E+09,9E+09,9E+09,9E+09,9E+09]];
    CONST jointtarget jB_t188 := [[44.9993,9.29655,-57.727,-0.000718084,2.53608,179.999],[9E+09,9E+09,9E+09,9E+09,9E+09,9E+09]];
    CONST jointtarget jBseed_t188 := [[44.9993,9.29655,-57.727,-0.000731559,2.53609,179.999],[9E+09,9E+09,9E+09,9E+09,9E+09,9E+09]];

    CONST robtarget rA_t192 := [[-54.6215,2798.58,2031.96],[0.634266,-0.31258,-0.502839,-0.497145],[1,1,-4,0],[9E+09,9E+09,9E+09,9E+09,9E+09,9E+09]];
    CONST robtarget rB_t192 := [[1716.76,-1818.08,2274.11],[0.544616,0.450827,0.604595,-0.366898],[-1,-1,-4,0],[9E+09,9E+09,9E+09,9E+09,9E+09,9E+09]];
    CONST robtarget rB_t192_c2 := [[1716.76,-1818.08,2274.11],[0.544616,0.450827,0.604595,-0.366898],[0,0,-4,0],[9E+09,9E+09,9E+09,9E+09,9E+09,9E+09]];
    CONST jointtarget jA_t192 := [[90,55.5943,-74.033,90,19.0912,-270],[9E+09,9E+09,9E+09,9E+09,9E+09,9E+09]];
    CONST jointtarget jB_t192 := [[-44.9992,34.8405,-54.4539,-44.9992,37.373,-314.999],[9E+09,9E+09,9E+09,9E+09,9E+09,9E+09]];
    CONST jointtarget jBseed_t192 := [[-44.9992,34.8405,-54.4539,-44.9992,37.373,-314.999],[9E+09,9E+09,9E+09,9E+09,9E+09,9E+09]];

    CONST robtarget rA_t194 := [[1591.57,0.0107639,1993.07],[0.708869,0.245423,0.592497,0.293631],[0,2,-2,0],[9E+09,9E+09,9E+09,9E+09,9E+09,9E+09]];
    CONST robtarget rB_t194 := [[96.2251,254.088,3271.92],[0.78246,-0.304432,0.472482,0.268028],[1,-1,4,0],[9E+09,9E+09,9E+09,9E+09,9E+09,9E+09]];
    CONST robtarget rB_t194_c5 := [[96.2251,254.088,3271.92],[0.78246,-0.304432,0.472482,0.268028],[0,0,0,0],[9E+09,9E+09,9E+09,9E+09,9E+09,9E+09]];
    CONST jointtarget jA_t194 := [[0.000393574,-22.6527,20.4309,180,7.99829,-135],[9E+09,9E+09,9E+09,9E+09,9E+09,9E+09]];
    CONST jointtarget jB_t194 := [[90.0004,-25.7363,-45.8684,-44.9996,54.5763,360],[9E+09,9E+09,9E+09,9E+09,9E+09,9E+09]];
    CONST jointtarget jBseed_t194 := [[90.0004,-25.7363,-45.8684,-44.9996,54.5763,360],[9E+09,9E+09,9E+09,9E+09,9E+09,9E+09]];

    CONST robtarget rA_t195 := [[96.2251,254.088,3271.92],[0.78246,-0.304432,0.472482,0.268028],[1,-1,4,0],[9E+09,9E+09,9E+09,9E+09,9E+09,9E+09]];
    CONST robtarget rB_t195 := [[1266.6,-1217.82,2896.72],[0.397424,-0.231823,0.320401,-0.828043],[-1,-3,-3,0],[9E+09,9E+09,9E+09,9E+09,9E+09,9E+09]];
    CONST robtarget rB_t195_c5 := [[1266.6,-1217.82,2896.72],[0.397424,-0.231823,0.320401,-0.828043],[0,0,0,0],[9E+09,9E+09,9E+09,9E+09,9E+09,9E+09]];
    CONST jointtarget jA_t195 := [[90.0004,-25.7363,-45.8684,-44.9996,54.5763,360],[9E+09,9E+09,9E+09,9E+09,9E+09,9E+09]];
    CONST jointtarget jB_t195 := [[-45.0008,6.22395,-38.6477,-225.001,16.9927,-225.001],[9E+09,9E+09,9E+09,9E+09,9E+09,9E+09]];
    CONST jointtarget jBseed_t195 := [[-45.0008,6.22395,-38.6477,-225.001,16.9927,-225.001],[9E+09,9E+09,9E+09,9E+09,9E+09,9E+09]];

    CONST robtarget rA_t197 := [[1069.37,1069.38,61.5578],[0.239594,0.686509,-0.686513,-1.51702E-7],[0,0,-1,0],[9E+09,9E+09,9E+09,9E+09,9E+09,9E+09]];
    CONST robtarget rB_t197 := [[2390.61,15.2187,412.458],[0.320235,-0.655845,0.632087,-0.260351],[0,1,-3,0],[9E+09,9E+09,9E+09,9E+09,9E+09,9E+09]];
    CONST robtarget rB_t197_c4 := [[2390.61,15.2187,412.458],[0.320235,-0.655845,0.632087,-0.260351],[0,-4,0,0],[9E+09,9E+09,9E+09,9E+09,9E+09,9E+09]];
    CONST jointtarget jA_t197 := [[45.0003,32.2367,39.5935,0.000333201,45.895,-44.9997],[9E+09,9E+09,9E+09,9E+09,9E+09,9E+09]];
    CONST jointtarget jB_t197 := [[0.000887153,41.2897,5.40634,135.001,7.3867,-224.999],[9E+09,9E+09,9E+09,9E+09,9E+09,9E+09]];
    CONST jointtarget jBseed_t197 := [[0.00088702,41.2897,5.40635,135.001,7.3867,-224.999],[9E+09,9E+09,9E+09,9E+09,9E+09,9E+09]];

    CONST robtarget rA_t198 := [[2390.61,15.2187,412.458],[0.320235,-0.655845,0.632087,-0.260351],[0,1,-3,0],[9E+09,9E+09,9E+09,9E+09,9E+09,9E+09]];
    CONST robtarget rB_t198 := [[971.585,-992.144,-144.851],[0.0614372,0.922725,0.379915,-0.0216647],[-1,-1,-2,0],[9E+09,9E+09,9E+09,9E+09,9E+09,9E+09]];
    CONST robtarget rB_t198_c2 := [[971.585,-992.144,-144.851],[0.0614372,0.922725,0.379915,-0.0216647],[0,0,-4,0],[9E+09,9E+09,9E+09,9E+09,9E+09,9E+09]];
    CONST robtarget rB_t198_c3 := [[971.585,-992.144,-144.851],[0.0614372,0.922725,0.379915,-0.0216647],[0,4,-4,0],[9E+09,9E+09,9E+09,9E+09,9E+09,9E+09]];
    CONST jointtarget jA_t198 := [[0.000887153,41.2897,5.40634,135.001,7.3867,-224.999],[9E+09,9E+09,9E+09,9E+09,9E+09,9E+09]];
    CONST jointtarget jB_t198 := [[-44.9998,38.9056,45.5327,-89.9998,4.99527,-180],[9E+09,9E+09,9E+09,9E+09,9E+09,9E+09]];
    CONST jointtarget jBseed_t198 := [[-44.9998,38.9056,45.5327,-89.9998,4.99527,-180],[9E+09,9E+09,9E+09,9E+09,9E+09,9E+09]];

    CONST robtarget rA_t200 := [[-96.1347,2841.92,1887.18],[0.459228,-0.00441754,-0.632801,-0.623421],[0,0,-4,0],[9E+09,9E+09,9E+09,9E+09,9E+09,9E+09]];
    CONST robtarget rB_t200 := [[1838.3,-1838.35,818.298],[0.713003,0.24335,0.587518,-0.295348],[-1,-3,1,0],[9E+09,9E+09,9E+09,9E+09,9E+09,9E+09]];
    CONST robtarget rB_t200_c2 := [[1838.3,-1838.35,818.298],[0.713003,0.24335,0.587518,-0.295348],[0,0,-4,0],[9E+09,9E+09,9E+09,9E+09,9E+09,9E+09]];
    CONST jointtarget jA_t200 := [[89.9999,56.8066,-70.8988,89.9999,35.1482,-315],[9E+09,9E+09,9E+09,9E+09,9E+09,9E+09]];
    CONST jointtarget jB_t200 := [[-45.0008,41.0663,-5.88885,-180.001,46.2007,179.999],[9E+09,9E+09,9E+09,9E+09,9E+09,9E+09]];
    CONST jointtarget jBseed_t200 := [[-45.0008,41.0663,-5.88885,-180.001,46.2007,179.999],[9E+09,9E+09,9E+09,9E+09,9E+09,9E+09]];

    CONST robtarget rA_t205 := [[1629.06,1609.53,189.691],[0.303834,-0.861411,0.370511,-0.168456],[0,2,0,0],[9E+09,9E+09,9E+09,9E+09,9E+09,9E+09]];
    CONST robtarget rB_t205 := [[1070.07,-1170.45,2076.59],[0.842518,0.461385,0.231331,-0.154187],[-1,-2,-2,0],[9E+09,9E+09,9E+09,9E+09,9E+09,9E+09]];
    CONST robtarget rB_t205_c6 := [[1070.07,-1170.45,2076.59],[0.842518,0.461385,0.231331,-0.154187],[0,4,0,0],[9E+09,9E+09,9E+09,9E+09,9E+09,9E+09]];
    CONST jointtarget jA_t205 := [[44.9994,45.3731,8.94924,224.999,6.70369,44.9993],[9E+09,9E+09,9E+09,9E+09,9E+09,9E+09]];
    CONST jointtarget jB_t205 := [[-44.9993,-20.9131,17.8521,-134.999,36.961,-179.999],[9E+09,9E+09,9E+09,9E+09,9E+09,9E+09]];
    CONST jointtarget jBseed_t205 := [[-44.9993,-20.9131,17.8521,-134.999,36.961,-179.999],[9E+09,9E+09,9E+09,9E+09,9E+09,9E+09]];

    CONST robtarget rA_t207 := [[-1040.33,1040.35,3262.83],[0.373608,-0.200178,0.0829138,0.901926],[1,-3,1,0],[9E+09,9E+09,9E+09,9E+09,9E+09,9E+09]];
    CONST robtarget rB_t207 := [[956.903,-9.53971,3259.97],[0.94867,0.0271598,0.31497,-0.0089962],[0,3,-3,0],[9E+09,9E+09,9E+09,9E+09,9E+09,9E+09]];
    CONST robtarget rB_t207_c5 := [[956.903,-9.53971,3259.97],[0.94867,0.0271598,0.31497,-0.0089962],[0,0,0,0],[9E+09,9E+09,9E+09,9E+09,9E+09,9E+09]];
    CONST jointtarget jA_t207 := [[134.999,17.9101,-72.3945,-180.001,10.4886,179.999],[9E+09,9E+09,9E+09,9E+09,9E+09,9E+09]];
    CONST jointtarget jB_t207 := [[0.000831477,-11.7502,-41.5162,270.001,3.27952,-269.999],[9E+09,9E+09,9E+09,9E+09,9E+09,9E+09]];
    CONST jointtarget jBseed_t207 := [[0.000831477,-11.7502,-41.5162,270.001,3.27952,-269.999],[9E+09,9E+09,9E+09,9E+09,9E+09,9E+09]];

    CONST robtarget rA_t208 := [[956.903,-9.53971,3259.97],[0.94867,0.0271598,0.31497,-0.0089962],[0,3,-3,0],[9E+09,9E+09,9E+09,9E+09,9E+09,9E+09]];
    CONST robtarget rB_t208 := [[-70.0194,2207.51,2313.39],[0.463849,-0.0127454,-0.472592,-0.749225],[0,1,-5,0],[9E+09,9E+09,9E+09,9E+09,9E+09,9E+09]];
    CONST robtarget rB_t208_c2 := [[-70.0194,2207.51,2313.39],[0.463849,-0.0127454,-0.472592,-0.749225],[0,0,-4,0],[9E+09,9E+09,9E+09,9E+09,9E+09,9E+09]];
    CONST jointtarget jA_t208 := [[0.000831477,-11.7502,-41.5162,270.001,3.27952,-269.999],[9E+09,9E+09,9E+09,9E+09,9E+09,9E+09]];
    CONST jointtarget jB_t208 := [[89.9998,14.3797,-24.3968,135,36.3713,-360],[9E+09,9E+09,9E+09,9E+09,9E+09,9E+09]];
    CONST jointtarget jBseed_t208 := [[89.9998,14.3797,-24.3968,135,36.3713,-360],[9E+09,9E+09,9E+09,9E+09,9E+09,9E+09]];

    CONST robtarget rA_t210 := [[1663.85,-1807.17,106.073],[0.656216,0.723698,-0.105426,0.185816],[-1,-2,3,0],[9E+09,9E+09,9E+09,9E+09,9E+09,9E+09]];
    CONST robtarget rB_t210 := [[2061.04,-48.8265,2409.91],[0.24275,-0.408195,0.295814,-0.82882],[-1,2,3,0],[9E+09,9E+09,9E+09,9E+09,9E+09,9E+09]];
    CONST robtarget rB_t210_c4 := [[2061.04,-48.8265,2409.91],[0.24275,-0.408195,0.295814,-0.82882],[0,-4,0,0],[9E+09,9E+09,9E+09,9E+09,9E+09,9E+09]];
    CONST robtarget rB_t210_c7 := [[2061.04,-48.8265,2409.91],[0.24275,-0.408195,0.295814,-0.82882],[0,-4,4,0],[9E+09,9E+09,9E+09,9E+09,9E+09,9E+09]];
    CONST jointtarget jA_t210 := [[-44.9995,57.7587,-2.92917,-134.999,59.1375,270.001],[9E+09,9E+09,9E+09,9E+09,9E+09,9E+09]];
    CONST jointtarget jB_t210 := [[-0.000990616,7.31895,-20.4731,224.999,24.405,359.999],[9E+09,9E+09,9E+09,9E+09,9E+09,9E+09]];
    CONST jointtarget jBseed_t210 := [[-0.000990722,7.31895,-20.473,224.999,24.405,359.999],[9E+09,9E+09,9E+09,9E+09,9E+09,9E+09]];

    CONST robtarget rA_t213 := [[1184.95,1138.28,213.19],[0.14362,-0.358402,0.921303,-0.0460686],[0,-1,-4,0],[9E+09,9E+09,9E+09,9E+09,9E+09,9E+09]];
    CONST robtarget rB_t213 := [[122.722,2561.17,1689.79],[0.0362535,0.508806,0.520109,0.685047],[0,-2,-2,0],[9E+09,9E+09,9E+09,9E+09,9E+09,9E+09]];
    CONST robtarget rB_t213_c2 := [[122.722,2561.17,1689.79],[0.0362535,0.508806,0.520109,0.685047],[0,0,-4,0],[9E+09,9E+09,9E+09,9E+09,9E+09,9E+09]];
    CONST jointtarget jA_t213 := [[45.0006,23.9601,41.24,-44.9994,16.2365,-314.999],[9E+09,9E+09,9E+09,9E+09,9E+09,9E+09]];
    CONST jointtarget jB_t213 := [[89.9998,30.5521,-25.5791,-90.0002,47.2921,-135],[9E+09,9E+09,9E+09,9E+09,9E+09,9E+09]];
    CONST jointtarget jBseed_t213 := [[89.9998,30.5521,-25.5791,-90.0002,47.2921,-135],[9E+09,9E+09,9E+09,9E+09,9E+09,9E+09]];

    CONST robtarget rA_t215 := [[-1743.32,-1709.81,2209.9],[0.237513,0.650339,0.209408,-0.690504],[-2,-1,0,0],[9E+09,9E+09,9E+09,9E+09,9E+09,9E+09]];
    CONST robtarget rB_t215 := [[97.6269,76.9328,2796.38],[0.0734141,-0.0458578,-0.234407,-0.968277],[-1,-3,-4,0],[9E+09,9E+09,9E+09,9E+09,9E+09,9E+09]];
    CONST robtarget rB_t215_c4 := [[97.6269,76.9328,2796.38],[0.0734141,-0.0458578,-0.234407,-0.968277],[0,-4,0,0],[9E+09,9E+09,9E+09,9E+09,9E+09,9E+09]];
    CONST jointtarget jA_t215 := [[-135,25.685,-37.767,-45.0004,11.5671,44.9996],[9E+09,9E+09,9E+09,9E+09,9E+09,9E+09]];
    CONST jointtarget jB_t215 := [[-3.3044E-5,-58.0114,2.79184,-225,40.6543,-315],[9E+09,9E+09,9E+09,9E+09,9E+09,9E+09]];
    CONST jointtarget jBseed_t215 := [[-3.62865E-5,-58.0114,2.79183,-225,40.6543,-315],[9E+09,9E+09,9E+09,9E+09,9E+09,9E+09]];

    CONST robtarget rA_t216 := [[97.6269,76.9328,2796.38],[0.0734141,-0.0458578,-0.234407,-0.968277],[-1,-3,-4,0],[9E+09,9E+09,9E+09,9E+09,9E+09,9E+09]];
    CONST robtarget rB_t216 := [[0.00100292,-1408.63,3151.17],[0.999676,-0.0254632,-3.25038E-7,1.07676E-6],[-1,-2,-1,0],[9E+09,9E+09,9E+09,9E+09,9E+09,9E+09]];
    CONST robtarget rB_t216_c4 := [[0.00100292,-1408.63,3151.17],[0.999676,-0.0254632,-3.25038E-7,1.07676E-6],[0,-4,0,0],[9E+09,9E+09,9E+09,9E+09,9E+09,9E+09]];
    CONST jointtarget jA_t216 := [[-3.3044E-5,-58.0114,2.79184,-225,40.6543,-315],[9E+09,9E+09,9E+09,9E+09,9E+09,9E+09]];
    CONST jointtarget jB_t216 := [[-90,5.03007,-47.8601,-180,50.0882,-90],[9E+09,9E+09,9E+09,9E+09,9E+09,9E+09]];
    CONST jointtarget jBseed_t216 := [[-90,5.03006,-47.86,-180,50.0882,-90],[9E+09,9E+09,9E+09,9E+09,9E+09,9E+09]];

    CONST robtarget rA_t217 := [[0.00100292,-1408.63,3151.17],[0.999676,-0.0254632,-3.25038E-7,1.07676E-6],[-1,-2,-1,0],[9E+09,9E+09,9E+09,9E+09,9E+09,9E+09]];
    CONST robtarget rB_t217 := [[2835.64,-51.6581,1273.4],[0.125303,0.671288,-0.0975797,0.723982],[0,2,-1,0],[9E+09,9E+09,9E+09,9E+09,9E+09,9E+09]];
    CONST robtarget rB_t217_c5 := [[2835.64,-51.6581,1273.4],[0.125303,0.671288,-0.0975797,0.723982],[0,0,0,0],[9E+09,9E+09,9E+09,9E+09,9E+09,9E+09]];
    CONST jointtarget jA_t217 := [[-90,5.03007,-47.8601,-180,50.0882,-90],[9E+09,9E+09,9E+09,9E+09,9E+09,9E+09]];
    CONST jointtarget jB_t217 := [[0.000678009,46.1788,-31.9904,225.001,25.9597,-44.9993],[9E+09,9E+09,9E+09,9E+09,9E+09,9E+09]];
    CONST jointtarget jBseed_t217 := [[0.000678091,46.1788,-31.9904,225.001,25.9597,-44.9993],[9E+09,9E+09,9E+09,9E+09,9E+09,9E+09]];

    CONST robtarget rA_t218 := [[2835.64,-51.6581,1273.4],[0.125303,0.671288,-0.0975797,0.723982],[0,2,-1,0],[9E+09,9E+09,9E+09,9E+09,9E+09,9E+09]];
    CONST robtarget rB_t218 := [[-97.2653,-2015.77,1876.56],[0.364885,0.11539,-0.88338,0.270524],[-2,-1,-2,0],[9E+09,9E+09,9E+09,9E+09,9E+09,9E+09]];
    CONST robtarget rB_t218_c5 := [[-97.2653,-2015.77,1876.56],[0.364885,0.11539,-0.88338,0.270524],[0,0,0,0],[9E+09,9E+09,9E+09,9E+09,9E+09,9E+09]];
    CONST jointtarget jA_t218 := [[0.000678009,46.1788,-31.9904,225.001,25.9597,-44.9993],[9E+09,9E+09,9E+09,9E+09,9E+09,9E+09]];
    CONST jointtarget jB_t218 := [[-90.001,2.69357,-2.17139,-45.001,55.4241,-90.001],[9E+09,9E+09,9E+09,9E+09,9E+09,9E+09]];
    CONST jointtarget jBseed_t218 := [[-90.001,2.69356,-2.17139,-45.001,55.4241,-90.001],[9E+09,9E+09,9E+09,9E+09,9E+09,9E+09]];

    CONST robtarget rA_t220 := [[64.2614,1589.31,2277.27],[0.405581,-0.0957962,0.629361,0.655921],[1,3,1,0],[9E+09,9E+09,9E+09,9E+09,9E+09,9E+09]];
    CONST robtarget rB_t220 := [[-942.211,942.213,2716.88],[0.980368,-0.139425,-0.139426,-1.06141E-6],[1,1,0,0],[9E+09,9E+09,9E+09,9E+09,9E+09,9E+09]];
    CONST robtarget rB_t220_c5 := [[-942.211,942.213,2716.88],[0.980368,-0.139425,-0.139426,-1.06141E-6],[0,0,0,0],[9E+09,9E+09,9E+09,9E+09,9E+09,9E+09]];
    CONST jointtarget jA_t220 := [[90.0003,-18.4814,6.63625,270,22.6344,135],[9E+09,9E+09,9E+09,9E+09,9E+09,9E+09]];
    CONST jointtarget jB_t220 := [[135,-19.2798,-5.73809,180,42.2382,45],[9E+09,9E+09,9E+09,9E+09,9E+09,9E+09]];
    CONST jointtarget jBseed_t220 := [[135,-19.2798,-5.73809,180,42.2382,44.9999],[9E+09,9E+09,9E+09,9E+09,9E+09,9E+09]];

    CONST robtarget rA_t221 := [[-942.211,942.213,2716.88],[0.980368,-0.139425,-0.139426,-1.06141E-6],[1,1,0,0],[9E+09,9E+09,9E+09,9E+09,9E+09,9E+09]];
    CONST robtarget rB_t221 := [[97.6801,352.927,2571.42],[0.942343,-0.0496091,0.303406,-0.132186],[1,2,-4,0],[9E+09,9E+09,9E+09,9E+09,9E+09,9E+09]];
    CONST robtarget rB_t221_c6 := [[97.6801,352.927,2571.42],[0.942343,-0.0496091,0.303406,-0.132186],[0,4,0,0],[9E+09,9E+09,9E+09,9E+09,9E+09,9E+09]];
    CONST jointtarget jA_t221 := [[135,-19.2798,-5.73809,180,42.2382,45],[9E+09,9E+09,9E+09,9E+09,9E+09,9E+09]];
    CONST jointtarget jB_t221 := [[90.0008,-59.6521,16.7412,225.001,55.8141,-314.999],[9E+09,9E+09,9E+09,9E+09,9E+09,9E+09]];
    CONST jointtarget jBseed_t221 := [[90.0008,-59.6521,16.7412,225.001,55.8141,-314.999],[9E+09,9E+09,9E+09,9E+09,9E+09,9E+09]];

    CONST robtarget rA_t224 := [[268.603,135.29,3003.22],[0.743266,-0.310339,0.393482,0.443189],[0,-3,3,0],[9E+09,9E+09,9E+09,9E+09,9E+09,9E+09]];
    CONST robtarget rB_t224 := [[1780.7,1697.48,2213.6],[0.460747,-0.61947,0.13909,-0.620179],[0,2,-1,0],[9E+09,9E+09,9E+09,9E+09,9E+09,9E+09]];
    CONST robtarget rB_t224_c8 := [[1780.7,1697.48,2213.6],[0.460747,-0.61947,0.13909,-0.620179],[0,0,4,0],[9E+09,9E+09,9E+09,9E+09,9E+09,9E+09]];
    CONST jointtarget jA_t224 := [[0.000699344,-42.1247,-15.97,-269.999,54.1057,315.001],[9E+09,9E+09,9E+09,9E+09,9E+09,9E+09]];
    CONST jointtarget jB_t224 := [[44.9997,27.3183,-39.2706,270,20.6275,-45.0002],[9E+09,9E+09,9E+09,9E+09,9E+09,9E+09]];
    CONST jointtarget jBseed_t224 := [[44.9997,27.3183,-39.2706,270,20.6275,-45.0003],[9E+09,9E+09,9E+09,9E+09,9E+09,9E+09]];

    CONST robtarget rA_t225 := [[1780.7,1697.48,2213.6],[0.460747,-0.61947,0.13909,-0.620179],[0,2,-1,0],[9E+09,9E+09,9E+09,9E+09,9E+09,9E+09]];
    CONST robtarget rB_t225 := [[-1082.32,1082.31,-339.715],[0.0722577,-0.994765,3.14028E-6,0.0722584],[1,2,1,0],[9E+09,9E+09,9E+09,9E+09,9E+09,9E+09]];
    CONST robtarget rB_t225_c5 := [[-1082.32,1082.31,-339.715],[0.0722577,-0.994765,3.14028E-6,0.0722584],[0,0,0,0],[9E+09,9E+09,9E+09,9E+09,9E+09,9E+09]];
    CONST jointtarget jA_t225 := [[44.9997,27.3183,-39.2706,270,20.6275,-45.0002],[9E+09,9E+09,9E+09,9E+09,9E+09,9E+09]];
    CONST jointtarget jB_t225 := [[135,52.1885,34.3962,180,8.31507,135],[9E+09,9E+09,9E+09,9E+09,9E+09,9E+09]];
    CONST jointtarget jBseed_t225 := [[135,52.1885,34.3962,180,8.31507,135],[9E+09,9E+09,9E+09,9E+09,9E+09,9E+09]];

    CONST robtarget rA_t227 := [[1614.34,-134.786,2923.24],[0.418326,0.000868129,0.570075,-0.707119],[-1,2,-1,0],[9E+09,9E+09,9E+09,9E+09,9E+09,9E+09]];
    CONST robtarget rB_t227 := [[-0.00661026,450.584,2707.86],[0.881598,-0.276264,0.114436,0.365194],[1,2,-3,0],[9E+09,9E+09,9E+09,9E+09,9E+09,9E+09]];
    CONST robtarget rB_t227_c2 := [[-0.00661026,450.584,2707.86],[0.881598,-0.276264,0.114436,0.365194],[0,0,-4,0],[9E+09,9E+09,9E+09,9E+09,9E+09,9E+09]];
    CONST jointtarget jA_t227 := [[-0.000949062,4.45143,-40.7941,269.999,53.798,-0.000947189],[9E+09,9E+09,9E+09,9E+09,9E+09,9E+09]];
    CONST jointtarget jB_t227 := [[90.0009,-54.0819,8.59615,180.001,9.71588,-224.999],[9E+09,9E+09,9E+09,9E+09,9E+09,9E+09]];
    CONST jointtarget jBseed_t227 := [[90.0009,-54.0819,8.59615,180.001,9.71587,-224.999],[9E+09,9E+09,9E+09,9E+09,9E+09,9E+09]];

    CONST robtarget rA_t228 := [[-0.00661026,450.584,2707.86],[0.881598,-0.276264,0.114436,0.365194],[1,2,-3,0],[9E+09,9E+09,9E+09,9E+09,9E+09,9E+09]];
    CONST robtarget rB_t228 := [[-1702.52,1842.64,2163.66],[0.736957,-0.356914,-0.189722,-0.541768],[1,2,3,0],[9E+09,9E+09,9E+09,9E+09,9E+09,9E+09]];
    CONST robtarget rB_t228_c5 := [[-1702.52,1842.64,2163.66],[0.736957,-0.356914,-0.189722,-0.541768],[0,0,0,0],[9E+09,9E+09,9E+09,9E+09,9E+09,9E+09]];
    CONST jointtarget jA_t228 := [[90.0009,-54.0819,8.59615,180.001,9.71588,-224.999],[9E+09,9E+09,9E+09,9E+09,9E+09,9E+09]];
    CONST jointtarget jB_t228 := [[134.999,33.5002,-42.7937,224.999,57.0061,314.999],[9E+09,9E+09,9E+09,9E+09,9E+09,9E+09]];
    CONST jointtarget jBseed_t228 := [[134.999,33.5002,-42.7937,224.999,57.0061,314.999],[9E+09,9E+09,9E+09,9E+09,9E+09,9E+09]];

    CONST robtarget rA_t229 := [[-1702.52,1842.64,2163.66],[0.736957,-0.356914,-0.189722,-0.541768],[1,2,3,0],[9E+09,9E+09,9E+09,9E+09,9E+09,9E+09]];
    CONST robtarget rB_t229 := [[100.772,178.842,3090.3],[0.0914845,0.333626,-0.102952,0.93259],[1,-2,-2,0],[9E+09,9E+09,9E+09,9E+09,9E+09,9E+09]];
    CONST robtarget rB_t229_c9 := [[100.772,178.842,3090.3],[0.0914845,0.333626,-0.102952,0.93259],[0,4,4,0],[9E+09,9E+09,9E+09,9E+09,9E+09,9E+09]];
    CONST jointtarget jA_t229 := [[134.999,33.5002,-42.7937,224.999,57.0061,314.999],[9E+09,9E+09,9E+09,9E+09,9E+09,9E+09]];
    CONST jointtarget jB_t229 := [[90.0005,-39.7589,-19.5685,-134.999,58.5809,-134.999],[9E+09,9E+09,9E+09,9E+09,9E+09,9E+09]];
    CONST jointtarget jBseed_t229 := [[90.0005,-39.7589,-19.5685,-134.999,58.5809,-134.999],[9E+09,9E+09,9E+09,9E+09,9E+09,9E+09]];

    CONST robtarget rA_t230 := [[100.772,178.842,3090.3],[0.0914845,0.333626,-0.102952,0.93259],[1,-2,-2,0],[9E+09,9E+09,9E+09,9E+09,9E+09,9E+09]];
    CONST robtarget rB_t230 := [[1424.92,-1604.71,2303.54],[0.752898,0.652419,-0.0824491,0.0263682],[-1,-2,-3,0],[9E+09,9E+09,9E+09,9E+09,9E+09,9E+09]];
    CONST robtarget rB_t230_c5 := [[1424.92,-1604.71,2303.54],[0.752898,0.652419,-0.0824491,0.0263682],[0,0,0,0],[9E+09,9E+09,9E+09,9E+09,9E+09,9E+09]];
    CONST jointtarget jA_t230 := [[90.0005,-39.7589,-19.5685,-134.999,58.5809,-134.999],[9E+09,9E+09,9E+09,9E+09,9E+09,9E+09]];
    CONST jointtarget jB_t230 := [[-45.0004,12.6072,-24.6309,-90.0004,49.57,-180],[9E+09,9E+09,9E+09,9E+09,9E+09,9E+09]];
    CONST jointtarget jBseed_t230 := [[-45.0004,12.6072,-24.6309,-90.0004,49.57,-180],[9E+09,9E+09,9E+09,9E+09,9E+09,9E+09]];

    CONST robtarget rA_t231 := [[1424.92,-1604.71,2303.54],[0.752898,0.652419,-0.0824491,0.0263682],[-1,-2,-3,0],[9E+09,9E+09,9E+09,9E+09,9E+09,9E+09]];
    CONST robtarget rB_t231 := [[-837.359,-760.809,1740.59],[0.381514,-0.366163,-0.566066,0.632409],[-2,3,-4,0],[9E+09,9E+09,9E+09,9E+09,9E+09,9E+09]];
    CONST robtarget rB_t231_c5 := [[-837.359,-760.809,1740.59],[0.381514,-0.366163,-0.566066,0.632409],[0,0,0,0],[9E+09,9E+09,9E+09,9E+09,9E+09,9E+09]];
    CONST jointtarget jA_t231 := [[-45.0004,12.6072,-24.6309,-90.0004,49.57,-180],[9E+09,9E+09,9E+09,9E+09,9E+09,9E+09]];
    CONST jointtarget jB_t231 := [[-134.999,-50.8261,45.3066,270.001,18.9172,-359.999],[9E+09,9E+09,9E+09,9E+09,9E+09,9E+09]];
    CONST jointtarget jBseed_t231 := [[-134.999,-50.8261,45.3066,270.001,18.9172,-359.999],[9E+09,9E+09,9E+09,9E+09,9E+09,9E+09]];

    CONST robtarget rA_t234 := [[-0.0209509,-1743.6,2641.73],[0.333459,0.187725,0.453218,-0.805082],[-2,1,1,0],[9E+09,9E+09,9E+09,9E+09,9E+09,9E+09]];
    CONST robtarget rB_t234 := [[1013.04,870.957,3214.61],[0.938615,0.243286,0.213605,-0.119108],[0,2,-4,0],[9E+09,9E+09,9E+09,9E+09,9E+09,9E+09]];
    CONST robtarget rB_t234_c2 := [[1013.04,870.957,3214.61],[0.938615,0.243286,0.213605,-0.119108],[0,0,-4,0],[9E+09,9E+09,9E+09,9E+09,9E+09,9E+09]];
    CONST jointtarget jA_t234 := [[-90.0007,-3.97167,-18.1402,179.999,9.13357,134.999],[9E+09,9E+09,9E+09,9E+09,9E+09,9E+09]];
    CONST jointtarget jB_t234 := [[44.9992,9.21597,-58.7466,224.999,58.2806,-270.001],[9E+09,9E+09,9E+09,9E+09,9E+09,9E+09]];
    CONST jointtarget jBseed_t234 := [[44.9992,9.21598,-58.7466,224.999,58.2806,-270.001],[9E+09,9E+09,9E+09,9E+09,9E+09,9E+09]];

    CONST robtarget rA_t235 := [[1013.04,870.957,3214.61],[0.938615,0.243286,0.213605,-0.119108],[0,2,-4,0],[9E+09,9E+09,9E+09,9E+09,9E+09,9E+09]];
    CONST robtarget rB_t235 := [[37.8488,-1631.05,3164.15],[0.330713,0.192521,-0.184506,0.905275],[-1,1,-3,0],[9E+09,9E+09,9E+09,9E+09,9E+09,9E+09]];
    CONST robtarget rB_t235_c2 := [[37.8488,-1631.05,3164.15],[0.330713,0.192521,-0.184506,0.905275],[0,0,-4,0],[9E+09,9E+09,9E+09,9E+09,9E+09,9E+09]];
    CONST robtarget rB_t235_c5 := [[37.8488,-1631.05,3164.15],[0.330713,0.192521,-0.184506,0.905275],[0,0,0,0],[9E+09,9E+09,9E+09,9E+09,9E+09,9E+09]];
    CONST jointtarget jA_t235 := [[44.9992,9.21597,-58.7466,224.999,58.2806,-270.001],[9E+09,9E+09,9E+09,9E+09,9E+09,9E+09]];
    CONST jointtarget jB_t235 := [[-89.9993,18.3898,-66.6656,135.001,18.6846,-269.999],[9E+09,9E+09,9E+09,9E+09,9E+09,9E+09]];
    CONST jointtarget jBseed_t235 := [[-89.9993,18.3898,-66.6656,135.001,18.6847,-269.999],[9E+09,9E+09,9E+09,9E+09,9E+09,9E+09]];

    CONST robtarget rA_t236 := [[37.8488,-1631.05,3164.15],[0.330713,0.192521,-0.184506,0.905275],[-1,1,-3,0],[9E+09,9E+09,9E+09,9E+09,9E+09,9E+09]];
    CONST robtarget rB_t236 := [[971.864,-924.841,1944.57],[0.514621,0.596902,0.0739999,0.611062],[-1,1,-1,0],[9E+09,9E+09,9E+09,9E+09,9E+09,9E+09]];
    CONST robtarget rB_t236_c2 := [[971.864,-924.841,1944.57],[0.514621,0.596902,0.0739999,0.611062],[0,0,-4,0],[9E+09,9E+09,9E+09,9E+09,9E+09,9E+09]];
    CONST jointtarget jA_t236 := [[-89.9993,18.3898,-66.6656,135.001,18.6846,-269.999],[9E+09,9E+09,9E+09,9E+09,9E+09,9E+09]];
    CONST jointtarget jB_t236 := [[-45.0009,-36.2322,31.5754,134.999,16.3646,-0.000886422],[9E+09,9E+09,9E+09,9E+09,9E+09,9E+09]];
    CONST jointtarget jBseed_t236 := [[-45.0009,-36.2322,31.5754,134.999,16.3646,-0.00089227],[9E+09,9E+09,9E+09,9E+09,9E+09,9E+09]];

    CONST robtarget rA_t237 := [[971.864,-924.841,1944.57],[0.514621,0.596902,0.0739999,0.611062],[-1,1,-1,0],[9E+09,9E+09,9E+09,9E+09,9E+09,9E+09]];
    CONST robtarget rB_t237 := [[1440.09,1440.05,1513.28],[0.342943,0.169833,0.410035,0.8279],[0,1,-2,0],[9E+09,9E+09,9E+09,9E+09,9E+09,9E+09]];
    CONST robtarget rB_t237_c5 := [[1440.09,1440.05,1513.28],[0.342943,0.169833,0.410035,0.8279],[0,0,0,0],[9E+09,9E+09,9E+09,9E+09,9E+09,9E+09]];
    CONST jointtarget jA_t237 := [[-45.0009,-36.2322,31.5754,134.999,16.3646,-0.000886422],[9E+09,9E+09,9E+09,9E+09,9E+09,9E+09]];
    CONST jointtarget jB_t237 := [[44.9991,3.54686,17.7529,179.999,58.6047,-90.0009],[9E+09,9E+09,9E+09,9E+09,9E+09,9E+09]];
    CONST jointtarget jBseed_t237 := [[44.9991,3.54686,17.7529,179.999,58.6047,-90.0009],[9E+09,9E+09,9E+09,9E+09,9E+09,9E+09]];

    CONST robtarget rA_t238 := [[1440.09,1440.05,1513.28],[0.342943,0.169833,0.410035,0.8279],[0,1,-2,0],[9E+09,9E+09,9E+09,9E+09,9E+09,9E+09]];
    CONST robtarget rB_t238 := [[-1102.6,1157.38,894.945],[0.354987,-0.882108,-0.307816,0.0334535],[1,-1,3,0],[9E+09,9E+09,9E+09,9E+09,9E+09,9E+09]];
    CONST robtarget rB_t238_c5 := [[-1102.6,1157.38,894.945],[0.354987,-0.882108,-0.307816,0.0334535],[0,0,0,0],[9E+09,9E+09,9E+09,9E+09,9E+09,9E+09]];
    CONST jointtarget jA_t238 := [[44.9991,3.54686,17.7529,179.999,58.6047,-90.0009],[9E+09,9E+09,9E+09,9E+09,9E+09,9E+09]];
    CONST jointtarget jB_t238 := [[135.001,-9.89349,46.1476,-44.9995,19.1552,315.001],[9E+09,9E+09,9E+09,9E+09,9E+09,9E+09]];
    CONST jointtarget jBseed_t238 := [[135.001,-9.89349,46.1477,-44.9995,19.1552,315.001],[9E+09,9E+09,9E+09,9E+09,9E+09,9E+09]];

    CONST robtarget rA_t246 := [[1952.78,111.891,2234.62],[0.742887,-0.484435,0.458824,-0.0540461],[-1,-4,2,0],[9E+09,9E+09,9E+09,9E+09,9E+09,9E+09]];
    CONST robtarget rB_t246 := [[39.7275,-2281.25,1420.1],[0.312982,0.242148,0.768695,-0.502509],[-1,1,2,0],[9E+09,9E+09,9E+09,9E+09,9E+09,9E+09]];
    CONST robtarget rB_t246_c7 := [[39.7275,-2281.25,1420.1],[0.312982,0.242148,0.768695,-0.502509],[0,-4,4,0],[9E+09,9E+09,9E+09,9E+09,9E+09,9E+09]];
    CONST jointtarget jA_t246 := [[-0.000846294,0.470599,-8.9636,-270.001,42.0808,224.999],[9E+09,9E+09,9E+09,9E+09,9E+09,9E+09]];
    CONST jointtarget jB_t246 := [[-89.9997,14.1087,3.82335,90.0003,13.7571,225],[9E+09,9E+09,9E+09,9E+09,9E+09,9E+09]];
    CONST jointtarget jBseed_t246 := [[-89.9997,14.1087,3.82336,90.0003,13.7571,225],[9E+09,9E+09,9E+09,9E+09,9E+09,9E+09]];

    CONST robtarget rA_t247 := [[39.7275,-2281.25,1420.1],[0.312982,0.242148,0.768695,-0.502509],[-1,1,2,0],[9E+09,9E+09,9E+09,9E+09,9E+09,9E+09]];
    CONST robtarget rB_t247 := [[2095.6,-0.00815796,1850.57],[0.642323,-0.275063,0.664057,-0.266063],[-1,-3,-3,0],[9E+09,9E+09,9E+09,9E+09,9E+09,9E+09]];
    CONST robtarget rB_t247_c5 := [[2095.6,-0.00815796,1850.57],[0.642323,-0.275063,0.664057,-0.266063],[0,0,0,0],[9E+09,9E+09,9E+09,9E+09,9E+09,9E+09]];
    CONST jointtarget jA_t247 := [[-89.9997,14.1087,3.82335,90.0003,13.7571,225],[9E+09,9E+09,9E+09,9E+09,9E+09,9E+09]];
    CONST jointtarget jB_t247 := [[-0.000223775,2.54708,2.34748,-180,2.98837,-225],[9E+09,9E+09,9E+09,9E+09,9E+09,9E+09]];
    CONST jointtarget jBseed_t247 := [[-0.000223975,2.54708,2.34748,-180,2.98837,-225],[9E+09,9E+09,9E+09,9E+09,9E+09,9E+09]];

    CONST robtarget rA_t248 := [[2095.6,-0.00815796,1850.57],[0.642323,-0.275063,0.664057,-0.266063],[-1,-3,-3,0],[9E+09,9E+09,9E+09,9E+09,9E+09,9E+09]];
    CONST robtarget rB_t248 := [[-106.71,-106.711,3356.33],[0.982385,-0.132138,0.132135,1.12991E-5],[-2,-2,3,0],[9E+09,9E+09,9E+09,9E+09,9E+09,9E+09]];
    CONST robtarget rB_t248_c4 := [[-106.71,-106.711,3356.33],[0.982385,-0.132138,0.132135,1.12991E-5],[0,-4,0,0],[9E+09,9E+09,9E+09,9E+09,9E+09,9E+09]];
    CONST jointtarget jA_t248 := [[-0.000223775,2.54708,2.34748,-180,2.98837,-225],[9E+09,9E+09,9E+09,9E+09,9E+09,9E+09]];
    CONST jointtarget jB_t248 := [[-135,-25.0807,-43.9522,-180,42.5074,315],[9E+09,9E+09,9E+09,9E+09,9E+09,9E+09]];
    CONST jointtarget jBseed_t248 := [[-135,-25.0807,-43.9521,-180,42.5074,315],[9E+09,9E+09,9E+09,9E+09,9E+09,9E+09]];

    CONST robtarget rA_t250 := [[-1310.11,1310.1,2158.6],[0.749831,-0.223565,-0.53973,-0.310587],[1,2,0,0],[9E+09,9E+09,9E+09,9E+09,9E+09,9E+09]];
    CONST robtarget rB_t250 := [[1515.37,1563.47,2244.33],[0.488925,-0.0780695,0.644381,0.582778],[0,-4,-1,0],[9E+09,9E+09,9E+09,9E+09,9E+09,9E+09]];
    CONST robtarget rB_t250_c5 := [[1515.37,1563.47,2244.33],[0.488925,-0.0780695,0.644381,0.582778],[0,0,0,0],[9E+09,9E+09,9E+09,9E+09,9E+09,9E+09]];
    CONST robtarget rB_t250_c8 := [[1515.37,1563.47,2244.33],[0.488925,-0.0780695,0.644381,0.582778],[0,0,4,0],[9E+09,9E+09,9E+09,9E+09,9E+09,9E+09]];
    CONST jointtarget jA_t250 := [[135,-7.77673,3.08542,180,13.8157,0.000152655],[9E+09,9E+09,9E+09,9E+09,9E+09,9E+09]];
    CONST jointtarget jB_t250 := [[44.9992,10.311,-19.5605,-270.001,11.7631,-45.0008],[9E+09,9E+09,9E+09,9E+09,9E+09,9E+09]];
    CONST jointtarget jBseed_t250 := [[44.9992,10.311,-19.5605,-270.001,11.7631,-45.0008],[9E+09,9E+09,9E+09,9E+09,9E+09,9E+09]];

    CONST robtarget rA_t251 := [[1515.37,1563.47,2244.33],[0.488925,-0.0780695,0.644381,0.582778],[0,-4,-1,0],[9E+09,9E+09,9E+09,9E+09,9E+09,9E+09]];
    CONST robtarget rB_t251 := [[1721.16,-94.3615,3029.65],[0.239031,0.0271505,0.298833,-0.923486],[-1,-2,3,0],[9E+09,9E+09,9E+09,9E+09,9E+09,9E+09]];
    CONST robtarget rB_t251_c4 := [[1721.16,-94.3615,3029.65],[0.239031,0.0271505,0.298833,-0.923486],[0,-4,0,0],[9E+09,9E+09,9E+09,9E+09,9E+09,9E+09]];
    CONST jointtarget jA_t251 := [[44.9992,10.311,-19.5605,-270.001,11.7631,-45.0008],[9E+09,9E+09,9E+09,9E+09,9E+09,9E+09]];
    CONST jointtarget jB_t251 := [[-0.000685878,17.4377,-57.7786,-135.001,53.0271,359.999],[9E+09,9E+09,9E+09,9E+09,9E+09,9E+09]];
    CONST jointtarget jBseed_t251 := [[-0.000685842,17.4377,-57.7786,-135.001,53.0271,359.999],[9E+09,9E+09,9E+09,9E+09,9E+09,9E+09]];

    CONST robtarget rA_t252 := [[1721.16,-94.3615,3029.65],[0.239031,0.0271505,0.298833,-0.923486],[-1,-2,3,0],[9E+09,9E+09,9E+09,9E+09,9E+09,9E+09]];
    CONST robtarget rB_t252 := [[265.678,-281.53,3513.71],[0.707743,0.0552923,-0.0334579,0.703508],[-1,-2,-2,0],[9E+09,9E+09,9E+09,9E+09,9E+09,9E+09]];
    CONST robtarget rB_t252_c7 := [[265.678,-281.53,3513.71],[0.707743,0.0552923,-0.0334579,0.703508],[0,-4,4,0],[9E+09,9E+09,9E+09,9E+09,9E+09,9E+09]];
    CONST jointtarget jA_t252 := [[-0.000685878,17.4377,-57.7786,-135.001,53.0271,359.999],[9E+09,9E+09,9E+09,9E+09,9E+09,9E+09]];
    CONST jointtarget jB_t252 := [[-45.0004,-1.45937,-78.3456,-135,5.44571,-90.0005],[9E+09,9E+09,9E+09,9E+09,9E+09,9E+09]];
    CONST jointtarget jBseed_t252 := [[-45.0004,-1.45939,-78.3456,-135,5.44572,-90.0004],[9E+09,9E+09,9E+09,9E+09,9E+09,9E+09]];

    CONST robtarget rA_t254 := [[-1639.36,1639.42,2615.76],[0.497168,1.21502E-6,-0.711071,-0.497195],[1,-1,1,0],[9E+09,9E+09,9E+09,9E+09,9E+09,9E+09]];
    CONST robtarget rB_t254 := [[105.801,2786.8,1555.48],[0.499121,-0.724193,-0.0517725,-0.473015],[0,2,3,0],[9E+09,9E+09,9E+09,9E+09,9E+09,9E+09]];
    CONST robtarget rB_t254_c5 := [[105.801,2786.8,1555.48],[0.499121,-0.724193,-0.0517725,-0.473015],[0,0,0,0],[9E+09,9E+09,9E+09,9E+09,9E+09,9E+09]];
    CONST robtarget rB_t254_c8 := [[105.801,2786.8,1555.48],[0.499121,-0.724193,-0.0517725,-0.473015],[0,0,4,0],[9E+09,9E+09,9E+09,9E+09,9E+09,9E+09]];
    CONST jointtarget jA_t254 := [[134.999,38.3892,-74.3067,-0.00091448,36.5618,134.999],[9E+09,9E+09,9E+09,9E+09,9E+09,9E+09]];
    CONST jointtarget jB_t254 := [[89.9996,44.1536,-40.1315,270,39.303,315],[9E+09,9E+09,9E+09,9E+09,9E+09,9E+09]];
    CONST jointtarget jBseed_t254 := [[89.9996,44.1536,-40.1315,270,39.303,315],[9E+09,9E+09,9E+09,9E+09,9E+09,9E+09]];

    CONST robtarget rA_t261 := [[1524.39,22.0418,1287.8],[0.620781,-0.0376666,0.781181,0.054482],[0,-3,-2,0],[9E+09,9E+09,9E+09,9E+09,9E+09,9E+09]];
    CONST robtarget rB_t261 := [[-71.8543,-980.834,2016.48],[0.131255,-0.177285,-0.580405,0.783883],[-1,-1,4,0],[9E+09,9E+09,9E+09,9E+09,9E+09,9E+09]];
    CONST robtarget rB_t261_c5 := [[-71.8543,-980.834,2016.48],[0.131255,-0.177285,-0.580405,0.783883],[0,0,0,0],[9E+09,9E+09,9E+09,9E+09,9E+09,9E+09]];
    CONST jointtarget jA_t261 := [[0.000708565,-25.1173,45.7826,-224.999,10.7486,-134.999],[9E+09,9E+09,9E+09,9E+09,9E+09,9E+09]];
    CONST jointtarget jB_t261 := [[-89.9996,-53.917,36.9512,-89.9996,25.4872,360],[9E+09,9E+09,9E+09,9E+09,9E+09,9E+09]];
    CONST jointtarget jBseed_t261 := [[-89.9996,-53.917,36.9512,-89.9996,25.4872,360],[9E+09,9E+09,9E+09,9E+09,9E+09,9E+09]];

    CONST robtarget rA_t263 := [[112.557,-2108.58,-123.214],[0.353242,-0.0764753,0.911289,-0.197291],[-1,1,-2,0],[9E+09,9E+09,9E+09,9E+09,9E+09,9E+09]];
    CONST robtarget rB_t263 := [[1670.66,-1670.65,761.16],[0.290207,0.602228,-0.249452,0.700625],[-1,-2,0,0],[9E+09,9E+09,9E+09,9E+09,9E+09,9E+09]];
    CONST robtarget rB_t263_c2 := [[1670.66,-1670.65,761.16],[0.290207,0.602228,-0.249452,0.700625],[0,0,-4,0],[9E+09,9E+09,9E+09,9E+09,9E+09,9E+09]];
    CONST robtarget rB_t263_c5 := [[1670.66,-1670.65,761.16],[0.290207,0.602228,-0.249452,0.700625],[0,0,0,0],[9E+09,9E+09,9E+09,9E+09,9E+09,9E+09]];
    CONST jointtarget jA_t263 := [[-90,54.818,10.7505,90,42.3756,-180],[9E+09,9E+09,9E+09,9E+09,9E+09,9E+09]];
    CONST jointtarget jB_t263 := [[-44.9999,31.9181,9.98078,-180,50.5368,7.12526E-5],[9E+09,9E+09,9E+09,9E+09,9E+09,9E+09]];
    CONST jointtarget jBseed_t263 := [[-44.9999,31.9181,9.98077,-180,50.5368,7.20541E-5],[9E+09,9E+09,9E+09,9E+09,9E+09,9E+09]];

    CONST robtarget rA_t264 := [[1670.66,-1670.65,761.16],[0.290207,0.602228,-0.249452,0.700625],[-1,-2,0,0],[9E+09,9E+09,9E+09,9E+09,9E+09,9E+09]];
    CONST robtarget rB_t264 := [[1024.8,936.097,3267.59],[0.315507,-0.1803,0.12596,-0.923083],[0,2,-1,0],[9E+09,9E+09,9E+09,9E+09,9E+09,9E+09]];
    CONST robtarget rB_t264_c4 := [[1024.8,936.097,3267.59],[0.315507,-0.1803,0.12596,-0.923083],[0,-4,0,0],[9E+09,9E+09,9E+09,9E+09,9E+09,9E+09]];
    CONST jointtarget jA_t264 := [[-44.9999,31.9181,9.98078,-180,50.5368,7.12526E-5],[9E+09,9E+09,9E+09,9E+09,9E+09,9E+09]];
    CONST jointtarget jB_t264 := [[44.9997,13.6289,-66.7806,225,32.0811,-45.0003],[9E+09,9E+09,9E+09,9E+09,9E+09,9E+09]];
    CONST jointtarget jBseed_t264 := [[44.9997,13.629,-66.7806,225,32.0811,-45.0003],[9E+09,9E+09,9E+09,9E+09,9E+09,9E+09]];

    CONST robtarget rA_t265 := [[1024.8,936.097,3267.59],[0.315507,-0.1803,0.12596,-0.923083],[0,2,-1,0],[9E+09,9E+09,9E+09,9E+09,9E+09,9E+09]];
    CONST robtarget rB_t265 := [[-1494.59,1381.06,2523.77],[0.457203,-0.560542,-0.202281,0.660182],[1,1,-2,0],[9E+09,9E+09,9E+09,9E+09,9E+09,9E+09]];
    CONST robtarget rB_t265_c5 := [[-1494.59,1381.06,2523.77],[0.457203,-0.560542,-0.202281,0.660182],[0,0,0,0],[9E+09,9E+09,9E+09,9E+09,9E+09,9E+09]];
    CONST jointtarget jA_t265 := [[44.9997,13.6289,-66.7806,225,32.0811,-45.0003],[9E+09,9E+09,9E+09,9E+09,9E+09,9E+09]];
    CONST jointtarget jB_t265 := [[135.001,9.28191,-28.5745,90.0008,28.721,-134.999],[9E+09,9E+09,9E+09,9E+09,9E+09,9E+09]];
    CONST jointtarget jBseed_t265 := [[135.001,9.28191,-28.5745,90.0008,28.721,-134.999],[9E+09,9E+09,9E+09,9E+09,9E+09,9E+09]];

    CONST robtarget rA_t267 := [[-1232.94,-1286,753.942],[0.350578,0.913016,0.0445684,-0.203739],[-2,-3,3,0],[9E+09,9E+09,9E+09,9E+09,9E+09,9E+09]];
    CONST robtarget rB_t267 := [[-1830.39,-1830.41,1728.77],[0.934106,0.252432,-0.252437,7.01489E-6],[-2,2,-1,0],[9E+09,9E+09,9E+09,9E+09,9E+09,9E+09]];
    CONST robtarget rB_t267_c7 := [[-1830.39,-1830.41,1728.77],[0.934106,0.252432,-0.252437,7.01489E-6],[0,-4,4,0],[9E+09,9E+09,9E+09,9E+09,9E+09,9E+09]];
    CONST jointtarget jA_t267 := [[-134.999,4.27564,39.2563,-269.999,12.9752,315.001],[9E+09,9E+09,9E+09,9E+09,9E+09,9E+09]];
    CONST jointtarget jB_t267 := [[-135,32.2037,-24.3492,180,56.0228,-44.9996],[9E+09,9E+09,9E+09,9E+09,9E+09,9E+09]];
    CONST jointtarget jBseed_t267 := [[-135,32.2037,-24.3492,180,56.0228,-44.9996],[9E+09,9E+09,9E+09,9E+09,9E+09,9E+09]];

    CONST robtarget rA_t268 := [[-1830.39,-1830.41,1728.77],[0.934106,0.252432,-0.252437,7.01489E-6],[-2,2,-1,0],[9E+09,9E+09,9E+09,9E+09,9E+09,9E+09]];
    CONST robtarget rB_t268 := [[1649.22,-1616.83,-124.081],[0.320719,0.345489,0.879823,-0.060733],[-1,1,-2,0],[9E+09,9E+09,9E+09,9E+09,9E+09,9E+09]];
    CONST robtarget rB_t268_c5 := [[1649.22,-1616.83,-124.081],[0.320719,0.345489,0.879823,-0.060733],[0,0,0,0],[9E+09,9E+09,9E+09,9E+09,9E+09,9E+09]];
    CONST jointtarget jA_t268 := [[-135,32.2037,-24.3492,180,56.0228,-44.9996],[9E+09,9E+09,9E+09,9E+09,9E+09,9E+09]];
    CONST jointtarget jB_t268 := [[-44.9997,58.4142,2.14118,135,11.1808,-135],[9E+09,9E+09,9E+09,9E+09,9E+09,9E+09]];
    CONST jointtarget jBseed_t268 := [[-44.9997,58.4143,2.14118,135,11.1808,-135],[9E+09,9E+09,9E+09,9E+09,9E+09,9E+09]];

